u16gBackSpeedRailWayAxleToolValue := TO_UINT(((u16gBackSpeedRailWayAxle.Value - u16gBackSpeedRailWayAxle.AppScalingOffset) * u16gBackSpeedRailWayAxle.AppScalingDivisor / u16gBackSpeedRailWayAxle.AppScalingMultiplier * u16gBackSpeedRailWayAxle.ToolScalingMultiplier / u16gBackSpeedRailWayAxle.ToolScalingDivisor) + u16gBackSpeedRailWayAxle.ToolScalingOffset);

                  
END_GET
END_PROPERTY

PROPERTY u16gAvdvancePeriodToolValue : UINT
GET
                    IF u16gAvdvancePeriod.ToolScalingDivisor = 0 OR u16gAvdvancePeriod.AppScalingMultiplier = 0 THEN
	_MatchLog^.Error("Get u16gAvdvancePeriodToolValue", "Division by Zero!");
	RETURN;
END_IF

u16gAvdvancePeriodToolValue := TO_UINT(((u16gAvdvancePeriod.Value - u16gAvdvancePeriod.AppScalingOffset) * u16gAvdvancePeriod.AppScalingDivisor / u16gAvdvancePeriod.AppScalingMultiplier * u16gAvdvancePeriod.ToolScalingMultiplier / u16gAvdvancePeriod.ToolScalingDivisor) + u16gAvdvancePeriod.ToolScalingOffset);

                  
END_GET
END_PROPERTY

PROPERTY u16gPressureEfficiencyRateToolValue : UINT
GET
                    IF u16gPressureEfficiencyRate.ToolScalingDivisor = 0 OR u16gPressureEfficiencyRate.AppScalingMultiplier = 0 THEN
	_MatchLog^.Error("Get u16gPressureEfficiencyRateToolValue", "Division by Zero!");
	RETURN;
END_IF

u16gPressureEfficiencyRateToolValue := TO_UINT(((u16gPressureEfficiencyRate.Value - u16gPressureEfficiencyRate.AppScalingOffset) * u16gPressureEfficiencyRate.AppScalingDivisor / u16gPressureEfficiencyRate.AppScalingMultiplier * u16gPressureEfficiencyRate.ToolScalingMultiplier / u16gPressureEfficiencyRate.ToolScalingDivisor) + u16gPressureEfficiencyRate.ToolScalingOffset);

                  
END_GET
END_PROPERTY

METHOD InitializeCanSignals
                  u16gFrontSpeedRailWayAxle.AppScalingDivisor :=1;
u16gFrontSpeedRailWayAxle.AppScalingMultiplier :=1;
u16gFrontSpeedRailWayAxle.AppScalingOffset :=0;
u16gFrontSpeedRailWayAxle.AppUnit :="";
u16gFrontSpeedRailWayAxle.CanDefault :=0;
u16gFrontSpeedRailWayAxle.CanInit :=0;
u16gFrontSpeedRailWayAxle.CanMax :=VBasic.LibConst.U16_MAX;
u16gFrontSpeedRailWayAxle.CanMin :=VBasic.LibConst.U16_MIN;
u16gFrontSpeedRailWayAxle.CanUnit :="";
u16gFrontSpeedRailWayAxle.Description :="Front Speed Railway Axle in Km/h (A24)";
u16gFrontSpeedRailWayAxle.ErrorReaction := eErrorReaction.ERSIG_DFLT;
u16gFrontSpeedRailWayAxle.ReceiverAdress :=1;
u16gFrontSpeedRailWayAxle.ToolScalingDivisor :=1;
u16gFrontSpeedRailWayAxle.ToolScalingMultiplier :=1;
u16gFrontSpeedRailWayAxle.ToolScalingOffset :=0;
u16gFrontSpeedRailWayAxle.ToolUnit :="";

u16gBackSpeedRailWayAxle.AppScalingDivisor :=1;
u16gBackSpeedRailWayAxle.AppScalingMultiplier :=1;
u16gBackSpeedRailWayAxle.AppScalingOffset :=0;
u16gBackSpeedRailWayAxle.AppUnit :="";
u16gBackSpeedRailWayAxle.CanDefault :=0;
u16gBackSpeedRailWayAxle.CanInit :=0;
u16gBackSpeedRailWayAxle.CanMax :=VBasic.LibConst.U16_MAX;
u16gBackSpeedRailWayAxle.CanMin :=VBasic.LibConst.U16_MIN;
u16gBackSpeedRailWayAxle.CanUnit :="";
u16gBackSpeedRailWayAxle.Description :="Back Speed Railway Axle in Km/h";
u16gBackSpeedRailWayAxle.ErrorReaction := eErrorReaction.ERSIG_DFLT;
u16gBackSpeedRailWayAxle.ReceiverAdress :=1;
u16gBackSpeedRailWayAxle.ToolScalingDivisor :=1;
u16gBackSpeedRailWayAxle.ToolScalingMultiplier :=1;
u16gBackSpeedRailWayAxle.ToolScalingOffset :=0;
u16gBackSpeedRailWayAxle.ToolUnit :="";

u16gAvdvancePeriod.AppScalingDivisor :=1;
u16gAvdvancePeriod.AppScalingMultiplier :=1;
u16gAvdvancePeriod.AppScalingOffset :=0;
u16gAvdvancePeriod.AppUnit :="";
u16gAvdvancePeriod.CanDefault :=0;
u16gAvdvancePeriod.CanInit :=0;
u16gAvdvancePeriod.CanMax :=VBasic.LibConst.U16_MAX;
u16gAvdvancePeriod.CanMin :=VBasic.LibConst.U16_MIN;
u16gAvdvancePeriod.CanUnit :="";
u16gAvdvancePeriod.Description :="new signal";
u16gAvdvancePeriod.ErrorReaction := eErrorReaction.ERSIG_DFLT;
u16gAvdvancePeriod.ReceiverAdress :=1;
u16gAvdvancePeriod.ToolScalingDivisor :=1;
u16gAvdvancePeriod.ToolScalingMultiplier :=1;
u16gAvdvancePeriod.ToolScalingOffset :=0;
u16gAvdvancePeriod.ToolUnit :="";

u16gPressureEfficiencyRate.AppScalingDivisor :=1;
u16gPressureEfficiencyRate.AppScalingMultiplier :=1;
u16gPressureEfficiencyRate.AppScalingOffset :=0;
u16gPressureEfficiencyRate.AppUnit :="";
u16gPressureEfficiencyRate.CanDefault :=0;
u16gPressureEfficiencyRate.CanInit :=0;
u16gPressureEfficiencyRate.CanMax :=VBasic.LibConst.U16_MAX;
u16gPressureEfficiencyRate.CanMin :=VBasic.LibConst.U16_MIN;
u16gPressureEfficiencyRate.CanUnit :="";
u16gPressureEfficiencyRate.Description :="new signal";
u16gPressureEfficiencyRate.ErrorReaction := eErrorReaction.ERSIG_DFLT;
u16gPressureEfficiencyRate.ReceiverAdress :=1;
u16gPressureEfficiencyRate.ToolScalingDivisor :=1;
u16gPressureEfficiencyRate.ToolScalingMultiplier :=1;
u16gPressureEfficiencyRate.ToolScalingOffset :=0;
u16gPressureEfficiencyRate.ToolUnit :="";


                
END_METHOD
END_FUNCTION_BLOCK

FUNCTION_BLOCK Msg4C0SendToEvision7MessageClass EXTENDS CanReceiveMessageClass
  VAR_INPUT
    u16gForwardPumpCurrent : UInt16CanSignalClass;
    u16gBackwardPumpCurrent : UInt16CanSignalClass;
    i16gTrans1PressureSensorValue : Int16CanSignalClass;
    i16gTrans2PressureSensorValue : Int16CanSignalClass;
    Counter : UInt32CanSignalClass;
  END_VAR

            
          

METHOD SetData
  VAR_INPUT
    CanMsgPointer : POINTER TO CanMessageClass;
  END_VAR
                  IF IsValidPointer(canMsgPointer,'SetData') THEN
	SUPER^.SetData(CanMsgPointer);
	//Set the new data
	u16gForwardPumpCurrent.Value := canMsgPointer^.GetUint16(0);
	u16gBackwardPumpCurrent.Value := canMsgPointer^.GetUint16(16);
	i16gTrans1PressureSensorValue.Value := canMsgPointer^.GetInt16(32);
	i16gTrans2PressureSensorValue.Value := canMsgPointer^.GetInt16(48);
	//And increase the counter
	Counter.Value := CanMsgPointer^.Counter.Value;
END_IF

                
END_METHOD

PROPERTY u16gForwardPumpCurrentRawValue : UINT
GET
                    IF u16gForwardPumpCurrent.AppScalingMultiplier = 0 THEN
	_MatchLog^.Error("Get u16gForwardPumpCurrentRawValue", "Division by Zero!");
	RETURN;
End_IF

u16gForwardPumpCurrentRawValue := TO_UINT((u16gForwardPumpCurrent.Value - u16gForwardPumpCurrent.AppScalingOffset) * u16gForwardPumpCurrent.AppScalingDivisor / u16gForwardPumpCurrent.AppScalingMultiplier);

                  
END_GET
END_PROPERTY

PROPERTY u16gBackwardPumpCurrentRawValue : UINT
GET
                    IF u16gBackwardPumpCurrent.AppScalingMultiplier = 0 THEN
	_MatchLog^.Error("Get u16gBackwardPumpCurrentRawValue", "Division by Zero!");
	RETURN;
End_IF

u16gBackwardPumpCurrentRawValue := TO_UINT((u16gBackwardPumpCurrent.Value - u16gBackwardPumpCurrent.AppScalingOffset) * u16gBackwardPumpCurrent.AppScalingDivisor / u16gBackwardPumpCurrent.AppScalingMultiplier);

                  
END_GET
END_PROPERTY

PROPERTY i16gTrans1PressureSensorValueRawValue : INT
GET
                    IF i16gTrans1PressureSensorValue.AppScalingMultiplier = 0 THEN
	_MatchLog^.Error("Get i16gTrans1PressureSensorValueRawValue", "Division by Zero!");
	RETURN;
End_IF

i16gTrans1PressureSensorValueRawValue := TO_INT((i16gTrans1PressureSensorValue.Value - i16gTrans1PressureSensorValue.AppScalingOffset) * i16gTrans1PressureSensorValue.AppScalingDivisor / i16gTrans1PressureSensorValue.AppScalingMultiplier);

                  
END_GET
END_PROPERTY

PROPERTY i16gTrans2PressureSensorValueRawValue : INT
GET
                    IF i16gTrans2PressureSensorValue.AppScalingMultiplier = 0 THEN
	_MatchLog^.Error("Get i16gTrans2PressureSensorValueRawValue", "Division by Zero!");
	RETURN;
End_IF

i16gTrans2PressureSensorValueRawValue := TO_INT((i16gTrans2PressureSensorValue.Value - i16gTrans2PressureSensorValue.AppScalingOffset) * i16gTrans2PressureSensorValue.AppScalingDivisor / i16gTrans2PressureSensorValue.AppScalingMultiplier);

                  
END_GET
END_PROPERTY

PROPERTY u16gForwardPumpCurrentToolValue : UINT
GET
                    IF u16gForwardPumpCurrent.ToolScalingDivisor = 0 OR u16gForwardPumpCurrent.AppScalingMultiplier = 0 THEN
	_MatchLog^.Error("Get u16gForwardPumpCurrentToolValue", "Division by Zero!");
	RETURN;
END_IF

u16gForwardPumpCurrentToolValue := TO_UINT(((u16gForwardPumpCurrent.Value - u16gForwardPumpCurrent.AppScalingOffset) * u16gForwardPumpCurrent.AppScalingDivisor / u16gForwardPumpCurrent.AppScalingMultiplier * u16gForwardPumpCurrent.ToolScalingMultiplier / u16gForwardPumpCurrent.ToolScalingDivisor) + u16gForwardPumpCurrent.ToolScalingOffset);

                  
END_GET
END_PROPERTY

PROPERTY u16gBackwardPumpCurrentToolValue : UINT
GET
                    IF u16gBackwardPumpCurrent.ToolScalingDivisor = 0 OR u16gBackwardPumpCurrent.AppScalingMultiplier = 0 THEN
	_MatchLog^.Error("Get u16gBackwardPumpCurrentToolValue", "Division by Zero!");
	RETURN;
END_IF

u16gBackwardPumpCurrentToolValue := TO_UINT(((u16gBackwardPumpCurrent.Value - u16gBackwardPumpCurrent.AppScalingOffset) * u16gBackwardPumpCurrent.AppScalingDivisor / u16gBackwardPumpCurrent.AppScalingMultiplier * u16gBackwardPumpCurrent.ToolScalingMultiplier / u16gBackwardPumpCurrent.ToolScalingDivisor) + u16gBackwardPumpCurrent.ToolScalingOffset);

                  
END_GET
END_PROPERTY

PROPERTY i16gTrans1PressureSensorValueToolValue : INT
GET
                    IF i16gTrans1PressureSensorValue.ToolScalingDivisor = 0 OR i16gTrans1PressureSensorValue.AppScalingMultiplier = 0 THEN
	_MatchLog^.Error("Get i16gTrans1PressureSensorValueToolValue", "Division by Zero!");
	RETURN;
END_IF

i16gTrans1PressureSensorValueToolValue := TO_INT(((i16gTrans1PressureSensorValue.Value - i16gTrans1PressureSensorValue.AppScalingOffset) * i16gTrans1PressureSensorValue.AppScalingDivisor / i16gTrans1PressureSensorValue.AppScalingMultiplier * i16gTrans1PressureSensorValue.ToolScalingMultiplier / i16gTrans1PressureSensorValue.ToolScalingDivisor) + i16gTrans1PressureSensorValue.ToolScalingOffset);

                  
END_GET
END_PROPERTY

PROPERTY i16gTrans2PressureSensorValueToolValue : INT
GET
                    IF i16gTrans2PressureSensorValue.ToolScalingDivisor = 0 OR i16gTrans2PressureSensorValue.AppScalingMultiplier = 0 THEN
	_MatchLog^.Error("Get i16gTrans2PressureSensorValueToolValue", "Division by Zero!");
	RETURN;
END_IF

i16gTrans2PressureSensorValueToolValue := TO_INT(((i16gTrans2PressureSensorValue.Value - i16gTrans2PressureSensorValue.AppScalingOffset) * i16gTrans2PressureSensorValue.AppScalingDivisor / i16gTrans2PressureSensorValue.AppScalingMultiplier * i16gTrans2PressureSensorValue.ToolScalingMultiplier / i16gTrans2PressureSensorValue.ToolScalingDivisor) + i16gTrans2PressureSensorValue.ToolScalingOffset);

                  
END_GET
END_PROPERTY

METHOD InitializeCanSignals
                  u16gForwardPumpCurrent.AppScalingDivisor :=1;
u16gForwardPumpCurrent.AppScalingMultiplier :=1;
u16gForwardPumpCurrent.AppScalingOffset :=0;
u16gForwardPumpCurrent.AppUnit :="";
u16gForwardPumpCurrent.CanDefault :=0;
u16gForwardPumpCurrent.CanInit :=0;
u16gForwardPumpCurrent.CanMax :=VBasic.LibConst.U16_MAX;
u16gForwardPumpCurrent.CanMin :=VBasic.LibConst.U16_MIN;
u16gForwardPumpCurrent.CanUnit :="";
u16gForwardPumpCurrent.Description :="Pressure transmission 1";
u16gForwardPumpCurrent.ErrorReaction := eErrorReaction.ERSIG_DFLT;
u16gForwardPumpCurrent.ReceiverAdress :=1;
u16gForwardPumpCurrent.ToolScalingDivisor :=1;
u16gForwardPumpCurrent.ToolScalingMultiplier :=1;
u16gForwardPumpCurrent.ToolScalingOffset :=0;
u16gForwardPumpCurrent.ToolUnit :="";

u16gBackwardPumpCurrent.AppScalingDivisor :=1;
u16gBackwardPumpCurrent.AppScalingMultiplier :=1;
u16gBackwardPumpCurrent.AppScalingOffset :=0;
u16gBackwardPumpCurrent.AppUnit :="";
u16gBackwardPumpCurrent.CanDefault :=0;
u16gBackwardPumpCurrent.CanInit :=0;
u16gBackwardPumpCurrent.CanMax :=VBasic.LibConst.U16_MAX;
u16gBackwardPumpCurrent.CanMin :=VBasic.LibConst.U16_MIN;
u16gBackwardPumpCurrent.CanUnit :="";
u16gBackwardPumpCurrent.Description :="Pressure transmission 2";
u16gBackwardPumpCurrent.ErrorReaction := eErrorReaction.ERSIG_DFLT;
u16gBackwardPumpCurrent.ReceiverAdress :=1;
u16gBackwardPumpCurrent.ToolScalingDivisor :=1;
u16gBackwardPumpCurrent.ToolScalingMultiplier :=1;
u16gBackwardPumpCurrent.ToolScalingOffset :=0;
u16gBackwardPumpCurrent.ToolUnit :="";

i16gTrans1PressureSensorValue.AppScalingDivisor :=1;
i16gTrans1PressureSensorValue.AppScalingMultiplier :=1;
i16gTrans1PressureSensorValue.AppScalingOffset :=0;
i16gTrans1PressureSensorValue.AppUnit :="";
i16gTrans1PressureSensorValue.CanDefault :=0;
i16gTrans1PressureSensorValue.CanInit :=0;
i16gTrans1PressureSensorValue.CanMax :=VBasic.LibConst.I16_MAX;
i16gTrans1PressureSensorValue.CanMin :=VBasic.LibConst.I16_MIN;
i16gTrans1PressureSensorValue.CanUnit :="";
i16gTrans1PressureSensorValue.Description :="new signal";
i16gTrans1PressureSensorValue.ErrorReaction := eErrorReaction.ERSIG_DFLT;
i16gTrans1PressureSensorValue.ReceiverAdress :=1;
i16gTrans1PressureSensorValue.ToolScalingDivisor :=1;
i16gTrans1PressureSensorValue.ToolScalingMultiplier :=1;
i16gTrans1PressureSensorValue.ToolScalingOffset :=0;
i16gTrans1PressureSensorValue.ToolUnit :="";

i16gTrans2PressureSensorValue.AppScalingDivisor :=1;
i16gTrans2PressureSensorValue.AppScalingMultiplier :=1;
i16gTrans2PressureSensorValue.AppScalingOffset :=0;
i16gTrans2PressureSensorValue.AppUnit :="";
i16gTrans2PressureSensorValue.CanDefault :=0;
i16gTrans2PressureSensorValue.CanInit :=0;
i16gTrans2PressureSensorValue.CanMax :=VBasic.LibConst.I16_MAX;
i16gTrans2PressureSensorValue.CanMin :=VBasic.LibConst.I16_MIN;
i16gTrans2PressureSensorValue.CanUnit :="";
i16gTrans2PressureSensorValue.Description :="new signal";
i16gTrans2PressureSensorValue.ErrorReaction := eErrorReaction.ERSIG_DFLT;
i16gTrans2PressureSensorValue.ReceiverAdress :=1;
i16gTrans2PressureSensorValue.ToolScalingDivisor :=1;
i16gTrans2PressureSensorValue.ToolScalingMultiplier :=1;
i16gTrans2PressureSensorValue.ToolScalingOffset :=0;
i16gTrans2PressureSensorValue.ToolUnit :="";


                
END_METHOD
END_FUNCTION_BLOCK

FUNCTION_BLOCK Msg5C0SendToEvision7MessageClass EXTENDS CanReceiveMessageClass
  VAR_INPUT
    boAbutementNacelleTrackSide : BoolCanSignalClass;
    boAbutementNacelleCenteredSide : BoolCanSignalClass;
    boBasketTurretLimitation : BoolCanSignalClass;
    boPin217Fault : BoolCanSignalClass;
    boPin230Fault : BoolCanSignalClass;
    boPin243Fault : BoolCanSignalClass;
    boPin244Fault : BoolCanSignalClass;
    boPin245Fault : BoolCanSignalClass;
    boPin256Fault : BoolCanSignalClass;
    boPin257Fault : BoolCanSignalClass;
    boPin258Fault : BoolCanSignalClass;
    boPin103Fault : BoolCanSignalClass;
    boPin127Fault : BoolCanSignalClass;
    boPin104Fault : BoolCanSignalClass;
    boPin128Fault : BoolCanSignalClass;
    boPin105Fault : BoolCanSignalClass;
    boPin129Fault : BoolCanSignalClass;
    boPin106Fault : BoolCanSignalClass;
    boPin130Fault : BoolCanSignalClass;
    boPin107Fault : BoolCanSignalClass;
    boPin131Fault : BoolCanSignalClass;
    boPin108Fault : BoolCanSignalClass;
    boPin132Fault : BoolCanSignalClass;
    boPin109Fault : BoolCanSignalClass;
    boPin133Fault : BoolCanSignalClass;
    boPin110Fault : BoolCanSignalClass;
    boPin134Fault : BoolCanSignalClass;
    boPin111Fault : BoolCanSignalClass;
    boPin135Fault : BoolCanSignalClass;
    boPin112Fault : BoolCanSignalClass;
    boPin136Fault : BoolCanSignalClass;
    boPin113Fault : BoolCanSignalClass;
    boPin137Fault : BoolCanSignalClass;
    boPin114Fault : BoolCanSignalClass;
    boPin138Fault : BoolCanSignalClass;
    boPin115Fault : BoolCanSignalClass;
    boPin139Fault : BoolCanSignalClass;
    boPin116Fault : BoolCanSignalClass;
    boPin140Fault : BoolCanSignalClass;
    boPin117Fault : BoolCanSignalClass;
    boPin141Fault : BoolCanSignalClass;
    boPin122Fault : BoolCanSignalClass;
    boPin146Fault : BoolCanSignalClass;
    boPin123Fault : BoolCanSignalClass;
    boPin147Fault : BoolCanSignalClass;
    boPin124Fault : BoolCanSignalClass;
    boPin148Fault : BoolCanSignalClass;
    boPin153Fault : BoolCanSignalClass;
    boPin177Fault : BoolCanSignalClass;
    boPin156Fault : BoolCanSignalClass;
    boPin180Fault : BoolCanSignalClass;
    boPin159Fault : BoolCanSignalClass;
    boPin183Fault : BoolCanSignalClass;
    boPin186Fault : BoolCanSignalClass;
    boPin162Fault : BoolCanSignalClass;
    boPin189Fault : BoolCanSignalClass;
    boPin165Fault : BoolCanSignalClass;
    boPin192Fault : BoolCanSignalClass;
    boPin168Fault : BoolCanSignalClass;
    boPin195Fault : BoolCanSignalClass;
    boPin171Fault : BoolCanSignalClass;
    boPin154Fault : BoolCanSignalClass;
    boPin178Fault : BoolCanSignalClass;
    boPin157Fault : BoolCanSignalClass;
    Counter : UInt32CanSignalClass;
  END_VAR

            
          

METHOD SetData
  VAR_INPUT
    CanMsgPointer : POINTER TO CanMessageClass;
  END_VAR
                  IF IsValidPointer(canMsgPointer,'SetData') THEN
	SUPER^.SetData(CanMsgPointer);
	//Set the new data
	boAbutementNacelleTrackSide.Value := canMsgPointer^.GetBoolOnBit(0);
	boAbutementNacelleCenteredSide.Value := canMsgPointer^.GetBoolOnBit(1);
	boBasketTurretLimitation.Value := canMsgPointer^.GetBoolOnBit(2);
	boPin217Fault.Value := canMsgPointer^.GetBoolOnBit(3);
	boPin230Fault.Value := canMsgPointer^.GetBoolOnBit(4);
	boPin243Fault.Value := canMsgPointer^.GetBoolOnBit(5);
	boPin244Fault.Value := canMsgPointer^.GetBoolOnBit(6);
	boPin245Fault.Value := canMsgPointer^.GetBoolOnBit(7);
	boPin256Fault.Value := canMsgPointer^.GetBoolOnBit(8);
	boPin257Fault.Value := canMsgPointer^.GetBoolOnBit(9);
	boPin258Fault.Value := canMsgPointer^.GetBoolOnBit(10);
	boPin103Fault.Value := canMsgPointer^.GetBoolOnBit(11);
	boPin127Fault.Value := canMsgPointer^.GetBoolOnBit(12);
	boPin104Fault.Value := canMsgPointer^.GetBoolOnBit(13);
	boPin128Fault.Value := canMsgPointer^.GetBoolOnBit(14);
	boPin105Fault.Value := canMsgPointer^.GetBoolOnBit(15);
	boPin129Fault.Value := canMsgPointer^.GetBoolOnBit(16);
	boPin106Fault.Value := canMsgPointer^.GetBoolOnBit(17);
	boPin130Fault.Value := canMsgPointer^.GetBoolOnBit(18);
	boPin107Fault.Value := canMsgPointer^.GetBoolOnBit(19);
	boPin131Fault.Value := canMsgPointer^.GetBoolOnBit(20);
	boPin108Fault.Value := canMsgPointer^.GetBoolOnBit(21);
	boPin132Fault.Value := canMsgPointer^.GetBoolOnBit(22);
	boPin109Fault.Value := canMsgPointer^.GetBoolOnBit(23);
	boPin133Fault.Value := canMsgPointer^.GetBoolOnBit(24);
	boPin110Fault.Value := canMsgPointer^.GetBoolOnBit(25);
	boPin134Fault.Value := canMsgPointer^.GetBoolOnBit(26);
	boPin111Fault.Value := canMsgPointer^.GetBoolOnBit(27);
	boPin135Fault.Value := canMsgPointer^.GetBoolOnBit(28);
	boPin112Fault.Value := canMsgPointer^.GetBoolOnBit(29);
	boPin136Fault.Value := canMsgPointer^.GetBoolOnBit(30);
	boPin113Fault.Value := canMsgPointer^.GetBoolOnBit(31);
	boPin137Fault.Value := canMsgPointer^.GetBoolOnBit(32);
	boPin114Fault.Value := canMsgPointer^.GetBoolOnBit(33);
	boPin138Fault.Value := canMsgPointer^.GetBoolOnBit(34);
	boPin115Fault.Value := canMsgPointer^.GetBoolOnBit(35);
	boPin139Fault.Value := canMsgPointer^.GetBoolOnBit(36);
	boPin116Fault.Value := canMsgPointer^.GetBoolOnBit(37);
	boPin140Fault.Value := canMsgPointer^.GetBoolOnBit(38);
	boPin117Fault.Value := canMsgPointer^.GetBoolOnBit(39);
	boPin141Fault.Value := canMsgPointer^.GetBoolOnBit(40);
	boPin122Fault.Value := canMsgPointer^.GetBoolOnBit(41);
	boPin146Fault.Value := canMsgPointer^.GetBoolOnBit(42);
	boPin123Fault.Value := canMsgPointer^.GetBoolOnBit(43);
	boPin147Fault.Value := canMsgPointer^.GetBoolOnBit(44);
	boPin124Fault.Value := canMsgPointer^.GetBoolOnBit(45);
	boPin148Fault.Value := canMsgPointer^.GetBoolOnBit(46);
	boPin153Fault.Value := canMsgPointer^.GetBoolOnBit(47);
	boPin177Fault.Value := canMsgPointer^.GetBoolOnBit(48);
	boPin156Fault.Value := canMsgPointer^.GetBoolOnBit(49);
	boPin180Fault.Value := canMsgPointer^.GetBoolOnBit(50);
	boPin159Fault.Value := canMsgPointer^.GetBoolOnBit(51);
	boPin183Fault.Value := canMsgPointer^.GetBoolOnBit(52);
	boPin186Fault.Value := canMsgPointer^.GetBoolOnBit(53);
	boPin162Fault.Value := canMsgPointer^.GetBoolOnBit(54);
	boPin189Fault.Value := canMsgPointer^.GetBoolOnBit(55);
	boPin165Fault.Value := canMsgPointer^.GetBoolOnBit(56);
	boPin192Fault.Value := canMsgPointer^.GetBoolOnBit(57);
	boPin168Fault.Value := canMsgPointer^.GetBoolOnBit(58);
	boPin195Fault.Value := canMsgPointer^.GetBoolOnBit(59);
	boPin171Fault.Value := canMsgPointer^.GetBoolOnBit(60);
	boPin154Fault.Value := canMsgPointer^.GetBoolOnBit(61);
	boPin178Fault.Value := canMsgPointer^.GetBoolOnBit(62);
	boPin157Fault.Value := canMsgPointer^.GetBoolOnBit(63);
	//And increase the counter
	Counter.Value := CanMsgPointer^.Counter.Value;
END_IF

                
END_METHOD

PROPERTY boAbutementNacelleTrackSideRawValue : BOOL
GET
                    boAbutementNacelleTrackSideRawValue := boAbutementNacelleTrackSide.Value;

                  
END_GET
END_PROPERTY

PROPERTY boAbutementNacelleCenteredSideRawValue : BOOL
GET
                    boAbutementNacelleCenteredSideRawValue := boAbutementNacelleCenteredSide.Value;

                  
END_GET
END_PROPERTY

PROPERTY boBasketTurretLimitationRawValue : BOOL
GET
                    boBasketTurretLimitationRawValue := boBasketTurretLimitation.Value;

                  
END_GET
END_PROPERTY

PROPERTY boPin217FaultRawValue : BOOL
GET
                    boPin217FaultRawValue := boPin217Fault.Value;

                  
END_GET
END_PROPERTY

PROPERTY boPin230FaultRawValue : BOOL
GET
                    boPin230FaultRawValue := boPin230Fault.Value;

                  
END_GET
END_PROPERTY

PROPERTY boPin243FaultRawValue : BOOL
GET
                    boPin243FaultRawValue := boPin243Fault.Value;

                  
END_GET
END_PROPERTY

PROPERTY boPin244FaultRawValue : BOOL
GET
                    boPin244FaultRawValue := boPin244Fault.Value;

                  
END_GET
END_PROPERTY

PROPERTY boPin245FaultRawValue : BOOL
GET
                    boPin245FaultRawValue := boPin245Fault.Value;

                  
END_GET
END_PROPERTY

PROPERTY boPin256FaultRawValue : BOOL
GET
                    boPin256FaultRawValue := boPin256Fault.Value;

                  
END_GET
END_PROPERTY

PROPERTY boPin257FaultRawValue : BOOL
GET
                    boPin257FaultRawValue := boPin257Fault.Value;

                  
END_GET
END_PROPERTY

PROPERTY boPin258FaultRawValue : BOOL
GET
                    boPin258FaultRawValue := boPin258Fault.Value;

                  
END_GET
END_PROPERTY

PROPERTY boPin103FaultRawValue : BOOL
GET
                    boPin103FaultRawValue := boPin103Fault.Value;

                  
END_GET
END_PROPERTY

PROPERTY boPin127FaultRawValue : BOOL
GET
                    boPin127FaultRawValue := boPin127Fault.Value;

                  
END_GET
END_PROPERTY

PROPERTY boPin104FaultRawValue : BOOL
GET
                    boPin104FaultRawValue := boPin104Fault.Value;

                  
END_GET
END_PROPERTY

PROPERTY boPin128FaultRawValue : BOOL
GET
                    boPin128FaultRawValue := boPin128Fault.Value;

                  
END_GET
END_PROPERTY

PROPERTY boPin105FaultRawValue : BOOL
GET
                    boPin105FaultRawValue := boPin105Fault.Value;

                  
END_GET
END_PROPERTY

PROPERTY boPin129FaultRawValue : BOOL
GET
                    boPin129FaultRawValue := boPin129Fault.Value;

                  
END_GET
END_PROPERTY

PROPERTY boPin106FaultRawValue : BOOL
GET
                    boPin106FaultRawValue := boPin106Fault.Value;

                  
END_GET
END_PROPERTY

PROPERTY boPin130FaultRawValue : BOOL
GET
                    boPin130FaultRawValue := boPin130Fault.Value;

                  
END_GET
END_PROPERTY

PROPERTY boPin107FaultRawValue : BOOL
GET
                    boPin107FaultRawValue := boPin107Fault.Value;

                  
END_GET
END_PROPERTY

PROPERTY boPin131FaultRawValue : BOOL
GET
                    boPin131FaultRawValue := boPin131Fault.Value;

                  
END_GET
END_PROPERTY

PROPERTY boPin108FaultRawValue : BOOL
GET
                    boPin108FaultRawValue := boPin108Fault.Value;

                  
END_GET
END_PROPERTY

PROPERTY boPin132FaultRawValue : BOOL
GET
                    boPin132FaultRawValue := boPin132Fault.Value;

                  
END_GET
END_PROPERTY

PROPERTY boPin109FaultRawValue : BOOL
GET
                    boPin109FaultRawValue := boPin109Fault.Value;

                  
END_GET
END_PROPERTY

PROPERTY boPin133FaultRawValue : BOOL
GET
                    boPin133FaultRawValue := boPin133Fault.Value;

                  
END_GET
END_PROPERTY

PROPERTY boPin110FaultRawValue : BOOL
GET
                    boPin110FaultRawValue := boPin110Fault.Value;

                  
END_GET
END_PROPERTY

PROPERTY boPin134FaultRawValue : BOOL
GET
                    boPin134FaultRawValue := boPin134Fault.Value;

                  
END_GET
END_PROPERTY

PROPERTY boPin111FaultRawValue : BOOL
GET
                    boPin111FaultRawValue := boPin111Fault.Value;

                  
END_GET
END_PROPERTY

PROPERTY boPin135FaultRawValue : BOOL
GET
                    boPin135FaultRawValue := boPin135Fault.Value;

                  
END_GET
END_PROPERTY

PROPERTY boPin112FaultRawValue : BOOL
GET
                    boPin112FaultRawValue := boPin112Fault.Value;

                  
END_GET
END_PROPERTY

PROPERTY boPin136FaultRawValue : BOOL
GET
                    boPin136FaultRawValue := boPin136Fault.Value;

                  
END_GET
END_PROPERTY

PROPERTY boPin113FaultRawValue : BOOL
GET
                    boPin113FaultRawValue := boPin113Fault.Value;

                  
END_GET
END_PROPERTY

PROPERTY boPin137FaultRawValue : BOOL
GET
                    boPin137FaultRawValue := boPin137Fault.Value;

                  
END_GET
END_PROPERTY

PROPERTY boPin114FaultRawValue : BOOL
GET
                    boPin114FaultRawValue := boPin114Fault.Value;

                  
END_GET
END_PROPERTY

PROPERTY boPin138FaultRawValue : BOOL
GET
                    boPin138FaultRawValue := boPin138Fault.Value;

                  
END_GET
END_PROPERTY

PROPERTY boPin115FaultRawValue : BOOL
GET
                    boPin115FaultRawValue := boPin115Fault.Value;

                  
END_GET
END_PROPERTY

PROPERTY boPin139FaultRawValue : BOOL
GET
                    boPin139FaultRawValue := boPin139Fault.Value;

                  
END_GET
END_PROPERTY

PROPERTY boPin116FaultRawValue : BOOL
GET
                    boPin116FaultRawValue := boPin116Fault.Value;

                  
END_GET
END_PROPERTY

PROPERTY boPin140FaultRawValue : BOOL
GET
                    boPin140FaultRawValue := boPin140Fault.Value;

                  
END_GET
END_PROPERTY

PROPERTY boPin117FaultRawValue : BOOL
GET
                    boPin117FaultRawValue := boPin117Fault.Value;

                  
END_GET
END_PROPERTY

PROPERTY boPin141FaultRawValue : BOOL
GET
                    boPin141FaultRawValue := boPin141Fault.Value;

                  
END_GET
END_PROPERTY

PROPERTY boPin122FaultRawValue : BOOL
GET
                    boPin122FaultRawValue := boPin122Fault.Value;

                  
END_GET
END_PROPERTY

PROPERTY boPin146FaultRawValue : BOOL
GET
                    boPin146FaultRawValue := boPin146Fault.Value;

                  
END_GET
END_PROPERTY

PROPERTY boPin123FaultRawValue : BOOL
GET
                    boPin123FaultRawValue := boPin123Fault.Value;

                  
END_GET
END_PROPERTY

PROPERTY boPin147FaultRawValue : BOOL
GET
                    boPin147FaultRawValue := boPin147Fault.Value;

                  
END_GET
END_PROPERTY

PROPERTY boPin124FaultRawValue : BOOL
GET
                    boPin124FaultRawValue := boPin124Fault.Value;

                  
END_GET
END_PROPERTY

PROPERTY boPin148FaultRawValue : BOOL
GET
                    boPin148FaultRawValue := boPin148Fault.Value;

                  
END_GET
END_PROPERTY

PROPERTY boPin153FaultRawValue : BOOL
GET
                    boPin153FaultRawValue := boPin153Fault.Value;

                  
END_GET
END_PROPERTY

PROPERTY boPin177FaultRawValue : BOOL
GET
                    boPin177FaultRawValue := boPin177Fault.Value;

                  
END_GET
END_PROPERTY

PROPERTY boPin156FaultRawValue : BOOL
GET
                    boPin156FaultRawValue := boPin156Fault.Value;

                  
END_GET
END_PROPERTY

PROPERTY boPin180FaultRawValue : BOOL
GET
                    boPin180FaultRawValue := boPin180Fault.Value;

                  
END_GET
END_PROPERTY

PROPERTY boPin159FaultRawValue : BOOL
GET
                    boPin159FaultRawValue := boPin159Fault.Value;

                  
END_GET
END_PROPERTY

PROPERTY boPin183FaultRawValue : BOOL
GET
                    boPin183FaultRawValue := boPin183Fault.Value;

                  
END_GET
END_PROPERTY

PROPERTY boPin186FaultRawValue : BOOL
GET
                    boPin186FaultRawValue := boPin186Fault.Value;

                  
END_GET
END_PROPERTY

PROPERTY boPin162FaultRawValue : BOOL
GET
                    boPin162FaultRawValue := boPin162Fault.Value;

                  
END_GET
END_PROPERTY

PROPERTY boPin189FaultRawValue : BOOL
GET
                    boPin189FaultRawValue := boPin189Fault.Value;

                  
END_GET
END_PROPERTY

PROPERTY boPin165FaultRawValue : BOOL
GET
                    boPin165FaultRawValue := boPin165Fault.Value;

                  
END_GET
END_PROPERTY

PROPERTY boPin192FaultRawValue : BOOL
GET
                    boPin192FaultRawValue := boPin192Fault.Value;

                  
END_GET
END_PROPERTY

PROPERTY boPin168FaultRawValue : BOOL
GET
                    boPin168FaultRawValue := boPin168Fault.Value;

                  
END_GET
END_PROPERTY

PROPERTY boPin195FaultRawValue : BOOL
GET
                    boPin195FaultRawValue := boPin195Fault.Value;

                  
END_GET
END_PROPERTY

PROPERTY boPin171FaultRawValue : BOOL
GET
                    boPin171FaultRawValue := boPin171Fault.Value;

                  
END_GET
END_PROPERTY

PROPERTY boPin154FaultRawValue : BOOL
GET
                    boPin154FaultRawValue := boPin154Fault.Value;

                  
END_GET
END_PROPERTY

PROPERTY boPin178FaultRawValue : BOOL
GET
                    boPin178FaultRawValue := boPin178Fault.Value;

                  
END_GET
END_PROPERTY

PROPERTY boPin157FaultRawValue : BOOL
GET
                    boPin157FaultRawValue := boPin157Fault.Value;

                  
END_GET
END_PROPERTY

PROPERTY boAbutementNacelleTrackSideToolValue : BOOL
GET
                    boAbutementNacelleTrackSideToolValue := boAbutementNacelleTrackSide.Value;

                  
END_GET
END_PROPERTY

PROPERTY boAbutementNacelleCenteredSideToolValue : BOOL
GET
                    boAbutementNacelleCenteredSideToolValue := boAbutementNacelleCenteredSide.Value;

                  
END_GET
END_PROPERTY

PROPERTY boBasketTurretLimitationToolValue : BOOL
GET
                    boBasketTurretLimitationToolValue := boBasketTurretLimitation.Value;

                  
END_GET
END_PROPERTY

PROPERTY boPin217FaultToolValue : BOOL
GET
                    boPin217FaultToolValue := boPin217Fault.Value;

                  
END_GET
END_PROPERTY

PROPERTY boPin230FaultToolValue : BOOL
GET
                    boPin230FaultToolValue := boPin230Fault.Value;

                  
END_GET
END_PROPERTY

PROPERTY boPin243FaultToolValue : BOOL
GET
                    boPin243FaultToolValue := boPin243Fault.Value;

                  
END_GET
END_PROPERTY

PROPERTY boPin244FaultToolValue : BOOL
GET
                    boPin244FaultToolValue := boPin244Fault.Value;

                  
END_GET
END_PROPERTY

PROPERTY boPin245FaultToolValue : BOOL
GET
                    boPin245FaultToolValue := boPin245Fault.Value;

                  
END_GET
END_PROPERTY

PROPERTY boPin256FaultToolValue : BOOL
GET
                    boPin256FaultToolValue := boPin256Fault.Value;

                  
END_GET
END_PROPERTY

PROPERTY boPin257FaultToolValue : BOOL
GET
                    boPin257FaultToolValue := boPin257Fault.Value;

                  
END_GET
END_PROPERTY

PROPERTY boPin258FaultToolValue : BOOL
GET
                    boPin258FaultToolValue := boPin258Fault.Value;

                  
END_GET
END_PROPERTY

PROPERTY boPin103FaultToolValue : BOOL
GET
                    boPin103FaultToolValue := boPin103Fault.Value;

                  
END_GET
END_PROPERTY

PROPERTY boPin127FaultToolValue : BOOL
GET
                    boPin127FaultToolValue := boPin127Fault.Value;

                  
END_GET
END_PROPERTY

PROPERTY boPin104FaultToolValue : BOOL
GET
                    boPin104FaultToolValue := boPin104Fault.Value;

                  
END_GET
END_PROPERTY

PROPERTY boPin128FaultToolValue : BOOL
GET
                    boPin128FaultToolValue := boPin128Fault.Value;

                  
END_GET
END_PROPERTY

PROPERTY boPin105FaultToolValue : BOOL
GET
                    boPin105FaultToolValue := boPin105Fault.Value;

                  
END_GET
END_PROPERTY

PROPERTY boPin129FaultToolValue : BOOL
GET
                    boPin129FaultToolValue := boPin129Fault.Value;

                  
END_GET
END_PROPERTY

PROPERTY boPin106FaultToolValue : BOOL
GET
                    boPin106FaultToolValue := boPin106Fault.Value;

                  
END_GET
END_PROPERTY

PROPERTY boPin130FaultToolValue : BOOL
GET
                    boPin130FaultToolValue := boPin130Fault.Value;

                  
END_GET
END_PROPERTY

PROPERTY boPin107FaultToolValue : BOOL
GET
                    boPin107FaultToolValue := boPin107Fault.Value;

                  
END_GET
END_PROPERTY

PROPERTY boPin131FaultToolValue : BOOL
GET
                    boPin131FaultToolValue := boPin131Fault.Value;

                  
END_GET
END_PROPERTY

PROPERTY boPin108FaultToolValue : BOOL
GET
                    boPin108FaultToolValue := boPin108Fault.Value;

                  
END_GET
END_PROPERTY

PROPERTY boPin132FaultToolValue : BOOL
GET
                    boPin132FaultToolValue := boPin132Fault.Value;

                  
END_GET
END_PROPERTY

PROPERTY boPin109FaultToolValue : BOOL
GET
                    boPin109FaultToolValue := boPin109Fault.Value;

                  
END_GET
END_PROPERTY

PROPERTY boPin133FaultToolValue : BOOL
GET
                    boPin133FaultToolValue := boPin133Fault.Value;

                  
END_GET
END_PROPERTY

PROPERTY boPin110FaultToolValue : BOOL
GET
                    boPin110FaultToolValue := boPin110Fault.Value;

                  
END_GET
END_PROPERTY

PROPERTY boPin134FaultToolValue : BOOL
GET
                    boPin134FaultToolValue := boPin134Fault.Value;

                  
END_GET
END_PROPERTY

PROPERTY boPin111FaultToolValue : BOOL
GET
                    boPin111FaultToolValue := boPin111Fault.Value;

                  
END_GET
END_PROPERTY

PROPERTY boPin135FaultToolValue : BOOL
GET
                    boPin135FaultToolValue := boPin135Fault.Value;

                  
END_GET
END_PROPERTY

PROPERTY boPin112FaultToolValue : BOOL
GET
                    boPin112FaultToolValue := boPin112Fault.Value;

                  
END_GET
END_PROPERTY

PROPERTY boPin136FaultToolValue : BOOL
GET
                    boPin136FaultToolValue := boPin136Fault.Value;

                  
END_GET
END_PROPERTY

PROPERTY boPin113FaultToolValue : BOOL
GET
                    boPin113FaultToolValue := boPin113Fault.Value;

                  
END_GET
END_PROPERTY

PROPERTY boPin137FaultToolValue : BOOL
GET
                    boPin137FaultToolValue := boPin137Fault.Value;

                  
END_GET
END_PROPERTY

PROPERTY boPin114FaultToolValue : BOOL
GET
                    boPin114FaultToolValue := boPin114Fault.Value;

                  
END_GET
END_PROPERTY

PROPERTY boPin138FaultToolValue : BOOL
GET
                    boPin138FaultToolValue := boPin138Fault.Value;

                  
END_GET
END_PROPERTY

PROPERTY boPin115FaultToolValue : BOOL
GET
                    boPin115FaultToolValue := boPin115Fault.Value;

                  
END_GET
END_PROPERTY

PROPERTY boPin139FaultToolValue : BOOL
GET
                    boPin139FaultToolValue := boPin139Fault.Value;

                  
END_GET
END_PROPERTY

PROPERTY boPin116FaultToolValue : BOOL
GET
                    boPin116FaultToolValue := boPin116Fault.Value;

                  
END_GET
END_PROPERTY

PROPERTY boPin140FaultToolValue : BOOL
GET
                    boPin140FaultToolValue := boPin140Fault.Value;

                  
END_GET
END_PROPERTY

PROPERTY boPin117FaultToolValue : BOOL
GET
                    boPin117FaultToolValue := boPin117Fault.Value;

                  
END_GET
END_PROPERTY

PROPERTY boPin141FaultToolValue : BOOL
GET
                    boPin141FaultToolValue := boPin141Fault.Value;

                  
END_GET
END_PROPERTY

PROPERTY boPin122FaultToolValue : BOOL
GET
                    boPin122FaultToolValue := boPin122Fault.Value;

                  
END_GET
END_PROPERTY

PROPERTY boPin146FaultToolValue : BOOL
GET
                    boPin146FaultToolValue := boPin146Fault.Value;

                  
END_GET
END_PROPERTY

PROPERTY boPin123FaultToolValue : BOOL
GET
                    boPin123FaultToolValue := boPin123Fault.Value;

                  
END_GET
END_PROPERTY

PROPERTY boPin147FaultToolValue : BOOL
GET
                    boPin147FaultToolValue := boPin147Fault.Value;

                  
END_GET
END_PROPERTY

PROPERTY boPin124FaultToolValue : BOOL
GET
                    boPin124FaultToolValue := boPin124Fault.Value;

                  
END_GET
END_PROPERTY

PROPERTY boPin148FaultToolValue : BOOL
GET
                    boPin148FaultToolValue := boPin148Fault.Value;

                  
END_GET
END_PROPERTY

PROPERTY boPin153FaultToolValue : BOOL
GET
                    boPin153FaultToolValue := boPin153Fault.Value;

                  
END_GET
END_PROPERTY

PROPERTY boPin177FaultToolValue : BOOL
GET
                    boPin177FaultToolValue := boPin177Fault.Value;

                  
END_GET
END_PROPERTY

PROPERTY boPin156FaultToolValue : BOOL
GET
                    boPin156FaultToolValue := boPin156Fault.Value;

                  
END_GET
END_PROPERTY

PROPERTY boPin180FaultToolValue : BOOL
GET
                    boPin180FaultToolValue := boPin180Fault.Value;

                  
END_GET
END_PROPERTY

PROPERTY boPin159FaultToolValue : BOOL
GET
                    boPin159FaultToolValue := boPin159Fault.Value;

                  
END_GET
END_PROPERTY

PROPERTY boPin183FaultToolValue : BOOL
GET
                    boPin183FaultToolValue := boPin183Fault.Value;

                  
END_GET
END_PROPERTY

PROPERTY boPin186FaultToolValue : BOOL
GET
                    boPin186FaultToolValue := boPin186Fault.Value;

                  
END_GET
END_PROPERTY

PROPERTY boPin162FaultToolValue : BOOL
GET
                    boPin162FaultToolValue := boPin162Fault.Value;

                  
END_GET
END_PROPERTY

PROPERTY boPin189FaultToolValue : BOOL
GET
                    boPin189FaultToolValue := boPin189Fault.Value;

                  
END_GET
END_PROPERTY

PROPERTY boPin165FaultToolValue : BOOL
GET
                    boPin165FaultToolValue := boPin165Fault.Value;

                  
END_GET
END_PROPERTY

PROPERTY boPin192FaultToolValue : BOOL
GET
                    boPin192FaultToolValue := boPin192Fault.Value;

                  
END_GET
END_PROPERTY

PROPERTY boPin168FaultToolValue : BOOL
GET
                    boPin168FaultToolValue := boPin168Fault.Value;

                  
END_GET
END_PROPERTY

PROPERTY boPin195FaultToolValue : BOOL
GET
                    boPin195FaultToolValue := boPin195Fault.Value;

                  
END_GET
END_PROPERTY

PROPERTY boPin171FaultToolValue : BOOL
GET
                    boPin171FaultToolValue := boPin171Fault.Value;

                  
END_GET
END_PROPERTY

PROPERTY boPin154FaultToolValue : BOOL
GET
                    boPin154FaultToolValue := boPin154Fault.Value;

                  
END_GET
END_PROPERTY

PROPERTY boPin178FaultToolValue : BOOL
GET
                    boPin178FaultToolValue := boPin178Fault.Value;

                  
END_GET
END_PROPERTY

PROPERTY boPin157FaultToolValue : BOOL
GET
                    boPin157FaultToolValue := boPin157Fault.Value;

                  
END_GET
END_PROPERTY

METHOD InitializeCanSignals
                  boAbutementNacelleTrackSide.AppScalingDivisor :=1;
boAbutementNacelleTrackSide.AppScalingMultiplier :=1;
boAbutementNacelleTrackSide.AppScalingOffset :=0;
boAbutementNacelleTrackSide.AppUnit :="";
boAbutementNacelleTrackSide.CanDefault :=0;
boAbutementNacelleTrackSide.CanInit :=0;
boAbutementNacelleTrackSide.CanMax :=1;
boAbutementNacelleTrackSide.CanMin :=0;
boAbutementNacelleTrackSide.CanUnit :="";
boAbutementNacelleTrackSide.Description :="for the Neotec diag pages";
boAbutementNacelleTrackSide.ErrorReaction := eErrorReaction.ERSIG_DFLT;
boAbutementNacelleTrackSide.ReceiverAdress :=1;
boAbutementNacelleTrackSide.ToolScalingDivisor :=1;
boAbutementNacelleTrackSide.ToolScalingMultiplier :=1;
boAbutementNacelleTrackSide.ToolScalingOffset :=0;
boAbutementNacelleTrackSide.ToolUnit :="";

boAbutementNacelleCenteredSide.AppScalingDivisor :=1;
boAbutementNacelleCenteredSide.AppScalingMultiplier :=1;
boAbutementNacelleCenteredSide.AppScalingOffset :=0;
boAbutementNacelleCenteredSide.AppUnit :="";
boAbutementNacelleCenteredSide.CanDefault :=0;
boAbutementNacelleCenteredSide.CanInit :=0;
boAbutementNacelleCenteredSide.CanMax :=1;
boAbutementNacelleCenteredSide.CanMin :=0;
boAbutementNacelleCenteredSide.CanUnit :="";
boAbutementNacelleCenteredSide.Description :="for the Neotec diag pages";
boAbutementNacelleCenteredSide.ErrorReaction := eErrorReaction.ERSIG_DFLT;
boAbutementNacelleCenteredSide.ReceiverAdress :=1;
boAbutementNacelleCenteredSide.ToolScalingDivisor :=1;
boAbutementNacelleCenteredSide.ToolScalingMultiplier :=1;
boAbutementNacelleCenteredSide.ToolScalingOffset :=0;
boAbutementNacelleCenteredSide.ToolUnit :="";

boBasketTurretLimitation.AppScalingDivisor :=1;
boBasketTurretLimitation.AppScalingMultiplier :=1;
boBasketTurretLimitation.AppScalingOffset :=0;
boBasketTurretLimitation.AppUnit :="";
boBasketTurretLimitation.CanDefault :=0;
boBasketTurretLimitation.CanInit :=0;
boBasketTurretLimitation.CanMax :=1;
boBasketTurretLimitation.CanMin :=0;
boBasketTurretLimitation.CanUnit :="";
boBasketTurretLimitation.Description :="for the Neotec diag pages";
boBasketTurretLimitation.ErrorReaction := eErrorReaction.ERSIG_DFLT;
boBasketTurretLimitation.ReceiverAdress :=1;
boBasketTurretLimitation.ToolScalingDivisor :=1;
boBasketTurretLimitation.ToolScalingMultiplier :=1;
boBasketTurretLimitation.ToolScalingOffset :=0;
boBasketTurretLimitation.ToolUnit :="";

boPin217Fault.AppScalingDivisor :=1;
boPin217Fault.AppScalingMultiplier :=1;
boPin217Fault.AppScalingOffset :=0;
boPin217Fault.AppUnit :="";
boPin217Fault.CanDefault :=0;
boPin217Fault.CanInit :=0;
boPin217Fault.CanMax :=1;
boPin217Fault.CanMin :=0;
boPin217Fault.CanUnit :="";
boPin217Fault.Description :="for the Neotec diag pages";
boPin217Fault.ErrorReaction := eErrorReaction.ERSIG_DFLT;
boPin217Fault.ReceiverAdress :=1;
boPin217Fault.ToolScalingDivisor :=1;
boPin217Fault.ToolScalingMultiplier :=1;
boPin217Fault.ToolScalingOffset :=0;
boPin217Fault.ToolUnit :="";

boPin230Fault.AppScalingDivisor :=1;
boPin230Fault.AppScalingMultiplier :=1;
boPin230Fault.AppScalingOffset :=0;
boPin230Fault.AppUnit :="";
boPin230Fault.CanDefault :=0;
boPin230Fault.CanInit :=0;
boPin230Fault.CanMax :=1;
boPin230Fault.CanMin :=0;
boPin230Fault.CanUnit :="";
boPin230Fault.Description :="for the Neotec diag pages";
boPin230Fault.ErrorReaction := eErrorReaction.ERSIG_DFLT;
boPin230Fault.ReceiverAdress :=1;
boPin230Fault.ToolScalingDivisor :=1;
boPin230Fault.ToolScalingMultiplier :=1;
boPin230Fault.ToolScalingOffset :=0;
boPin230Fault.ToolUnit :="";

boPin243Fault.AppScalingDivisor :=1;
boPin243Fault.AppScalingMultiplier :=1;
boPin243Fault.AppScalingOffset :=0;
boPin243Fault.AppUnit :="";
boPin243Fault.CanDefault :=0;
boPin243Fault.CanInit :=0;
boPin243Fault.CanMax :=1;
boPin243Fault.CanMin :=0;
boPin243Fault.CanUnit :="";
boPin243Fault.Description :="for the Neotec diag pages";
boPin243Fault.ErrorReaction := eErrorReaction.ERSIG_DFLT;
boPin243Fault.ReceiverAdress :=1;
boPin243Fault.ToolScalingDivisor :=1;
boPin243Fault.ToolScalingMultiplier :=1;
boPin243Fault.ToolScalingOffset :=0;
boPin243Fault.ToolUnit :="";

boPin244Fault.AppScalingDivisor :=1;
boPin244Fault.AppScalingMultiplier :=1;
boPin244Fault.AppScalingOffset :=0;
boPin244Fault.AppUnit :="";
boPin244Fault.CanDefault :=0;
boPin244Fault.CanInit :=0;
boPin244Fault.CanMax :=1;
boPin244Fault.CanMin :=0;
boPin244Fault.CanUnit :="";
boPin244Fault.Description :="for the Neotec diag pages";
boPin244Fault.ErrorReaction := eErrorReaction.ERSIG_DFLT;
boPin244Fault.ReceiverAdress :=1;
boPin244Fault.ToolScalingDivisor :=1;
boPin244Fault.ToolScalingMultiplier :=1;
boPin244Fault.ToolScalingOffset :=0;
boPin244Fault.ToolUnit :="";

boPin245Fault.AppScalingDivisor :=1;
boPin245Fault.AppScalingMultiplier :=1;
boPin245Fault.AppScalingOffset :=0;
boPin245Fault.AppUnit :="";
boPin245Fault.CanDefault :=0;
boPin245Fault.CanInit :=0;
boPin245Fault.CanMax :=1;
boPin245Fault.CanMin :=0;
boPin245Fault.CanUnit :="";
boPin245Fault.Description :="for the Neotec diag pages";
boPin245Fault.ErrorReaction := eErrorReaction.ERSIG_DFLT;
boPin245Fault.ReceiverAdress :=1;
boPin245Fault.ToolScalingDivisor :=1;
boPin245Fault.ToolScalingMultiplier :=1;
boPin245Fault.ToolScalingOffset :=0;
boPin245Fault.ToolUnit :="";

boPin256Fault.AppScalingDivisor :=1;
boPin256Fault.AppScalingMultiplier :=1;
boPin256Fault.AppScalingOffset :=0;
boPin256Fault.AppUnit :="";
boPin256Fault.CanDefault :=0;
boPin256Fault.CanInit :=0;
boPin256Fault.CanMax :=1;
boPin256Fault.CanMin :=0;
boPin256Fault.CanUnit :="";
boPin256Fault.Description :="for the Neotec diag pages";
boPin256Fault.ErrorReaction := eErrorReaction.ERSIG_DFLT;
boPin256Fault.ReceiverAdress :=1;
boPin256Fault.ToolScalingDivisor :=1;
boPin256Fault.ToolScalingMultiplier :=1;
boPin256Fault.ToolScalingOffset :=0;
boPin256Fault.ToolUnit :="";

boPin257Fault.AppScalingDivisor :=1;
boPin257Fault.AppScalingMultiplier :=1;
boPin257Fault.AppScalingOffset :=0;
boPin257Fault.AppUnit :="";
boPin257Fault.CanDefault :=0;
boPin257Fault.CanInit :=0;
boPin257Fault.CanMax :=1;
boPin257Fault.CanMin :=0;
boPin257Fault.CanUnit :="";
boPin257Fault.Description :="for the Neotec diag pages";
boPin257Fault.ErrorReaction := eErrorReaction.ERSIG_DFLT;
boPin257Fault.ReceiverAdress :=1;
boPin257Fault.ToolScalingDivisor :=1;
boPin257Fault.ToolScalingMultiplier :=1;
boPin257Fault.ToolScalingOffset :=0;
boPin257Fault.ToolUnit :="";

boPin258Fault.AppScalingDivisor :=1;
boPin258Fault.AppScalingMultiplier :=1;
boPin258Fault.AppScalingOffset :=0;
boPin258Fault.AppUnit :="";
boPin258Fault.CanDefault :=0;
boPin258Fault.CanInit :=0;
boPin258Fault.CanMax :=1;
boPin258Fault.CanMin :=0;
boPin258Fault.CanUnit :="";
boPin258Fault.Description :="for the Neotec diag pages";
boPin258Fault.ErrorReaction := eErrorReaction.ERSIG_DFLT;
boPin258Fault.ReceiverAdress :=1;
boPin258Fault.ToolScalingDivisor :=1;
boPin258Fault.ToolScalingMultiplier :=1;
boPin258Fault.ToolScalingOffset :=0;
boPin258Fault.ToolUnit :="";

boPin103Fault.AppScalingDivisor :=1;
boPin103Fault.AppScalingMultiplier :=1;
boPin103Fault.AppScalingOffset :=0;
boPin103Fault.AppUnit :="";
boPin103Fault.CanDefault :=0;
boPin103Fault.CanInit :=0;
boPin103Fault.CanMax :=1;
boPin103Fault.CanMin :=0;
boPin103Fault.CanUnit :="";
boPin103Fault.Description :="for the Neotec diag pages";
boPin103Fault.ErrorReaction := eErrorReaction.ERSIG_DFLT;
boPin103Fault.ReceiverAdress :=1;
boPin103Fault.ToolScalingDivisor :=1;
boPin103Fault.ToolScalingMultiplier :=1;
boPin103Fault.ToolScalingOffset :=0;
boPin103Fault.ToolUnit :="";

boPin127Fault.AppScalingDivisor :=1;
boPin127Fault.AppScalingMultiplier :=1;
boPin127Fault.AppScalingOffset :=0;
boPin127Fault.AppUnit :="";
boPin127Fault.CanDefault :=0;
boPin127Fault.CanInit :=0;
boPin127Fault.CanMax :=1;
boPin127Fault.CanMin :=0;
boPin127Fault.CanUnit :="";
boPin127Fault.Description :="for the Neotec diag pages";
boPin127Fault.ErrorReaction := eErrorReaction.ERSIG_DFLT;
boPin127Fault.ReceiverAdress :=1;
boPin127Fault.ToolScalingDivisor :=1;
boPin127Fault.ToolScalingMultiplier :=1;
boPin127Fault.ToolScalingOffset :=0;
boPin127Fault.ToolUnit :="";

boPin104Fault.AppScalingDivisor :=1;
boPin104Fault.AppScalingMultiplier :=1;
boPin104Fault.AppScalingOffset :=0;
boPin104Fault.AppUnit :="";
boPin104Fault.CanDefault :=0;
boPin104Fault.CanInit :=0;
boPin104Fault.CanMax :=1;
boPin104Fault.CanMin :=0;
boPin104Fault.CanUnit :="";
boPin104Fault.Description :="for the Neotec diag pages";
boPin104Fault.ErrorReaction := eErrorReaction.ERSIG_DFLT;
boPin104Fault.ReceiverAdress :=1;
boPin104Fault.ToolScalingDivisor :=1;
boPin104Fault.ToolScalingMultiplier :=1;
boPin104Fault.ToolScalingOffset :=0;
boPin104Fault.ToolUnit :="";

boPin128Fault.AppScalingDivisor :=1;
boPin128Fault.AppScalingMultiplier :=1;
boPin128Fault.AppScalingOffset :=0;
boPin128Fault.AppUnit :="";
boPin128Fault.CanDefault :=0;
boPin128Fault.CanInit :=0;
boPin128Fault.CanMax :=1;
boPin128Fault.CanMin :=0;
boPin128Fault.CanUnit :="";
boPin128Fault.Description :="for the Neotec diag pages";
boPin128Fault.ErrorReaction := eErrorReaction.ERSIG_DFLT;
boPin128Fault.ReceiverAdress :=1;
boPin128Fault.ToolScalingDivisor :=1;
boPin128Fault.ToolScalingMultiplier :=1;
boPin128Fault.ToolScalingOffset :=0;
boPin128Fault.ToolUnit :="";

boPin105Fault.AppScalingDivisor :=1;
boPin105Fault.AppScalingMultiplier :=1;
boPin105Fault.AppScalingOffset :=0;
boPin105Fault.AppUnit :="";
boPin105Fault.CanDefault :=0;
boPin105Fault.CanInit :=0;
boPin105Fault.CanMax :=1;
boPin105Fault.CanMin :=0;
boPin105Fault.CanUnit :="";
boPin105Fault.Description :="for the Neotec diag pages";
boPin105Fault.ErrorReaction := eErrorReaction.ERSIG_DFLT;
boPin105Fault.ReceiverAdress :=1;
boPin105Fault.ToolScalingDivisor :=1;
boPin105Fault.ToolScalingMultiplier :=1;
boPin105Fault.ToolScalingOffset :=0;
boPin105Fault.ToolUnit :="";

boPin129Fault.AppScalingDivisor :=1;
boPin129Fault.AppScalingMultiplier :=1;
boPin129Fault.AppScalingOffset :=0;
boPin129Fault.AppUnit :="";
boPin129Fault.CanDefault :=0;
boPin129Fault.CanInit :=0;
boPin129Fault.CanMax :=1;
boPin129Fault.CanMin :=0;
boPin129Fault.CanUnit :="";
boPin129Fault.Description :="for the Neotec diag pages";
boPin129Fault.ErrorReaction := eErrorReaction.ERSIG_DFLT;
boPin129Fault.ReceiverAdress :=1;
boPin129Fault.ToolScalingDivisor :=1;
boPin129Fault.ToolScalingMultiplier :=1;
boPin129Fault.ToolScalingOffset :=0;
boPin129Fault.ToolUnit :="";

boPin106Fault.AppScalingDivisor :=1;
boPin106Fault.AppScalingMultiplier :=1;
boPin106Fault.AppScalingOffset :=0;
boPin106Fault.AppUnit :="";
boPin106Fault.CanDefault :=0;
boPin106Fault.CanInit :=0;
boPin106Fault.CanMax :=1;
boPin106Fault.CanMin :=0;
boPin106Fault.CanUnit :="";
boPin106Fault.Description :="for the Neotec diag pages";
boPin106Fault.ErrorReaction := eErrorReaction.ERSIG_DFLT;
boPin106Fault.ReceiverAdress :=1;
boPin106Fault.ToolScalingDivisor :=1;
boPin106Fault.ToolScalingMultiplier :=1;
boPin106Fault.ToolScalingOffset :=0;
boPin106Fault.ToolUnit :="";

boPin130Fault.AppScalingDivisor :=1;
boPin130Fault.AppScalingMultiplier :=1;
boPin130Fault.AppScalingOffset :=0;
boPin130Fault.AppUnit :="";
boPin130Fault.CanDefault :=0;
boPin130Fault.CanInit :=0;
boPin130Fault.CanMax :=1;
boPin130Fault.CanMin :=0;
boPin130Fault.CanUnit :="";
boPin130Fault.Description :="for the Neotec diag pages";
boPin130Fault.ErrorReaction := eErrorReaction.ERSIG_DFLT;
boPin130Fault.ReceiverAdress :=1;
boPin130Fault.ToolScalingDivisor :=1;
boPin130Fault.ToolScalingMultiplier :=1;
boPin130Fault.ToolScalingOffset :=0;
boPin130Fault.ToolUnit :="";

boPin107Fault.AppScalingDivisor :=1;
boPin107Fault.AppScalingMultiplier :=1;
boPin107Fault.AppScalingOffset :=0;
boPin107Fault.AppUnit :="";
boPin107Fault.CanDefault :=0;
boPin107Fault.CanInit :=0;
boPin107Fault.CanMax :=1;
boPin107Fault.CanMin :=0;
boPin107Fault.CanUnit :="";
boPin107Fault.Description :="for the Neotec diag pages";
boPin107Fault.ErrorReaction := eErrorReaction.ERSIG_DFLT;
boPin107Fault.ReceiverAdress :=1;
boPin107Fault.ToolScalingDivisor :=1;
boPin107Fault.ToolScalingMultiplier :=1;
boPin107Fault.ToolScalingOffset :=0;
boPin107Fault.ToolUnit :="";

boPin131Fault.AppScalingDivisor :=1;
boPin131Fault.AppScalingMultiplier :=1;
boPin131Fault.AppScalingOffset :=0;
boPin131Fault.AppUnit :="";
boPin131Fault.CanDefault :=0;
boPin131Fault.CanInit :=0;
boPin131Fault.CanMax :=1;
boPin131Fault.CanMin :=0;
boPin131Fault.CanUnit :="";
boPin131Fault.Description :="for the Neotec diag pages";
boPin131Fault.ErrorReaction := eErrorReaction.ERSIG_DFLT;
boPin131Fault.ReceiverAdress :=1;
boPin131Fault.ToolScalingDivisor :=1;
boPin131Fault.ToolScalingMultiplier :=1;
boPin131Fault.ToolScalingOffset :=0;
boPin131Fault.ToolUnit :="";

boPin108Fault.AppScalingDivisor :=1;
boPin108Fault.AppScalingMultiplier :=1;
boPin108Fault.AppScalingOffset :=0;
boPin108Fault.AppUnit :="";
boPin108Fault.CanDefault :=0;
boPin108Fault.CanInit :=0;
boPin108Fault.CanMax :=1;
boPin108Fault.CanMin :=0;
boPin108Fault.CanUnit :="";
boPin108Fault.Description :="for the Neotec diag pages";
boPin108Fault.ErrorReaction := eErrorReaction.ERSIG_DFLT;
boPin108Fault.ReceiverAdress :=1;
boPin108Fault.ToolScalingDivisor :=1;
boPin108Fault.ToolScalingMultiplier :=1;
boPin108Fault.ToolScalingOffset :=0;
boPin108Fault.ToolUnit :="";

boPin132Fault.AppScalingDivisor :=1;
boPin132Fault.AppScalingMultiplier :=1;
boPin132Fault.AppScalingOffset :=0;
boPin132Fault.AppUnit :="";
boPin132Fault.CanDefault :=0;
boPin132Fault.CanInit :=0;
boPin132Fault.CanMax :=1;
boPin132Fault.CanMin :=0;
boPin132Fault.CanUnit :="";
boPin132Fault.Description :="for the Neotec diag pages";
boPin132Fault.ErrorReaction := eErrorReaction.ERSIG_DFLT;
boPin132Fault.ReceiverAdress :=1;
boPin132Fault.ToolScalingDivisor :=1;
boPin132Fault.ToolScalingMultiplier :=1;
boPin132Fault.ToolScalingOffset :=0;
boPin132Fault.ToolUnit :="";

boPin109Fault.AppScalingDivisor :=1;
boPin109Fault.AppScalingMultiplier :=1;
boPin109Fault.AppScalingOffset :=0;
boPin109Fault.AppUnit :="";
boPin109Fault.CanDefault :=0;
boPin109Fault.CanInit :=0;
boPin109Fault.CanMax :=1;
boPin109Fault.CanMin :=0;
boPin109Fault.CanUnit :="";
boPin109Fault.Description :="for the Neotec diag pages";
boPin109Fault.ErrorReaction := eErrorReaction.ERSIG_DFLT;
boPin109Fault.ReceiverAdress :=1;
boPin109Fault.ToolScalingDivisor :=1;
boPin109Fault.ToolScalingMultiplier :=1;
boPin109Fault.ToolScalingOffset :=0;
boPin109Fault.ToolUnit :="";

boPin133Fault.AppScalingDivisor :=1;
boPin133Fault.AppScalingMultiplier :=1;
boPin133Fault.AppScalingOffset :=0;
boPin133Fault.AppUnit :="";
boPin133Fault.CanDefault :=0;
boPin133Fault.CanInit :=0;
boPin133Fault.CanMax :=1;
boPin133Fault.CanMin :=0;
boPin133Fault.CanUnit :="";
boPin133Fault.Description :="for the Neotec diag pages";
boPin133Fault.ErrorReaction := eErrorReaction.ERSIG_DFLT;
boPin133Fault.ReceiverAdress :=1;
boPin133Fault.ToolScalingDivisor :=1;
boPin133Fault.ToolScalingMultiplier :=1;
boPin133Fault.ToolScalingOffset :=0;
boPin133Fault.ToolUnit :="";

boPin110Fault.AppScalingDivisor :=1;
boPin110Fault.AppScalingMultiplier :=1;
boPin110Fault.AppScalingOffset :=0;
boPin110Fault.AppUnit :="";
boPin110Fault.CanDefault :=0;
boPin110Fault.CanInit :=0;
boPin110Fault.CanMax :=1;
boPin110Fault.CanMin :=0;
boPin110Fault.CanUnit :="";
boPin110Fault.Description :="for the Neotec diag pages";
boPin110Fault.ErrorReaction := eErrorReaction.ERSIG_DFLT;
boPin110Fault.ReceiverAdress :=1;
boPin110Fault.ToolScalingDivisor :=1;
boPin110Fault.ToolScalingMultiplier :=1;
boPin110Fault.ToolScalingOffset :=0;
boPin110Fault.ToolUnit :="";

boPin134Fault.AppScalingDivisor :=1;
boPin134Fault.AppScalingMultiplier :=1;
boPin134Fault.AppScalingOffset :=0;
boPin134Fault.AppUnit :="";
boPin134Fault.CanDefault :=0;
boPin134Fault.CanInit :=0;
boPin134Fault.CanMax :=1;
boPin134Fault.CanMin :=0;
boPin134Fault.CanUnit :="";
boPin134Fault.Description :="for the Neotec diag pages";
boPin134Fault.ErrorReaction := eErrorReaction.ERSIG_DFLT;
boPin134Fault.ReceiverAdress :=1;
boPin134Fault.ToolScalingDivisor :=1;
boPin134Fault.ToolScalingMultiplier :=1;
boPin134Fault.ToolScalingOffset :=0;
boPin134Fault.ToolUnit :="";

boPin111Fault.AppScalingDivisor :=1;
boPin111Fault.AppScalingMultiplier :=1;
boPin111Fault.AppScalingOffset :=0;
boPin111Fault.AppUnit :="";
boPin111Fault.CanDefault :=0;
boPin111Fault.CanInit :=0;
boPin111Fault.CanMax :=1;
boPin111Fault.CanMin :=0;
boPin111Fault.CanUnit :="";
boPin111Fault.Description :="for the Neotec diag pages";
boPin111Fault.ErrorReaction := eErrorReaction.ERSIG_DFLT;
boPin111Fault.ReceiverAdress :=1;
boPin111Fault.ToolScalingDivisor :=1;
boPin111Fault.ToolScalingMultiplier :=1;
boPin111Fault.ToolScalingOffset :=0;
boPin111Fault.ToolUnit :="";

boPin135Fault.AppScalingDivisor :=1;
boPin135Fault.AppScalingMultiplier :=1;
boPin135Fault.AppScalingOffset :=0;
boPin135Fault.AppUnit :="";
boPin135Fault.CanDefault :=0;
boPin135Fault.CanInit :=0;
boPin135Fault.CanMax :=1;
boPin135Fault.CanMin :=0;
boPin135Fault.CanUnit :="";
boPin135Fault.Description :="for the Neotec diag pages";
boPin135Fault.ErrorReaction := eErrorReaction.ERSIG_DFLT;
boPin135Fault.ReceiverAdress :=1;
boPin135Fault.ToolScalingDivisor :=1;
boPin135Fault.ToolScalingMultiplier :=1;
boPin135Fault.ToolScalingOffset :=0;
boPin135Fault.ToolUnit :="";

boPin112Fault.AppScalingDivisor :=1;
boPin112Fault.AppScalingMultiplier :=1;
boPin112Fault.AppScalingOffset :=0;
boPin112Fault.AppUnit :="";
boPin112Fault.CanDefault :=0;
boPin112Fault.CanInit :=0;
boPin112Fault.CanMax :=1;
boPin112Fault.CanMin :=0;
boPin112Fault.CanUnit :="";
boPin112Fault.Description :="for the Neotec diag pages";
boPin112Fault.ErrorReaction := eErrorReaction.ERSIG_DFLT;
boPin112Fault.ReceiverAdress :=1;
boPin112Fault.ToolScalingDivisor :=1;
boPin112Fault.ToolScalingMultiplier :=1;
boPin112Fault.ToolScalingOffset :=0;
boPin112Fault.ToolUnit :="";

boPin136Fault.AppScalingDivisor :=1;
boPin136Fault.AppScalingMultiplier :=1;
boPin136Fault.AppScalingOffset :=0;
boPin136Fault.AppUnit :="";
boPin136Fault.CanDefault :=0;
boPin136Fault.CanInit :=0;
boPin136Fault.CanMax :=1;
boPin136Fault.CanMin :=0;
boPin136Fault.CanUnit :="";
boPin136Fault.Description :="for the Neotec diag pages";
boPin136Fault.ErrorReaction := eErrorReaction.ERSIG_DFLT;
boPin136Fault.ReceiverAdress :=1;
boPin136Fault.ToolScalingDivisor :=1;
boPin136Fault.ToolScalingMultiplier :=1;
boPin136Fault.ToolScalingOffset :=0;
boPin136Fault.ToolUnit :="";

boPin113Fault.AppScalingDivisor :=1;
boPin113Fault.AppScalingMultiplier :=1;
boPin113Fault.AppScalingOffset :=0;
boPin113Fault.AppUnit :="";
boPin113Fault.CanDefault :=0;
boPin113Fault.CanInit :=0;
boPin113Fault.CanMax :=1;
boPin113Fault.CanMin :=0;
boPin113Fault.CanUnit :="";
boPin113Fault.Description :="for the Neotec diag pages";
boPin113Fault.ErrorReaction := eErrorReaction.ERSIG_DFLT;
boPin113Fault.ReceiverAdress :=1;
boPin113Fault.ToolScalingDivisor :=1;
boPin113Fault.ToolScalingMultiplier :=1;
boPin113Fault.ToolScalingOffset :=0;
boPin113Fault.ToolUnit :="";

boPin137Fault.AppScalingDivisor :=1;
boPin137Fault.AppScalingMultiplier :=1;
boPin137Fault.AppScalingOffset :=0;
boPin137Fault.AppUnit :="";
boPin137Fault.CanDefault :=0;
boPin137Fault.CanInit :=0;
boPin137Fault.CanMax :=1;
boPin137Fault.CanMin :=0;
boPin137Fault.CanUnit :="";
boPin137Fault.Description :="for the Neotec diag pages";
boPin137Fault.ErrorReaction := eErrorReaction.ERSIG_DFLT;
boPin137Fault.ReceiverAdress :=1;
boPin137Fault.ToolScalingDivisor :=1;
boPin137Fault.ToolScalingMultiplier :=1;
boPin137Fault.ToolScalingOffset :=0;
boPin137Fault.ToolUnit :="";

boPin114Fault.AppScalingDivisor :=1;
boPin114Fault.AppScalingMultiplier :=1;
boPin114Fault.AppScalingOffset :=0;
boPin114Fault.AppUnit :="";
boPin114Fault.CanDefault :=0;
boPin114Fault.CanInit :=0;
boPin114Fault.CanMax :=1;
boPin114Fault.CanMin :=0;
boPin114Fault.CanUnit :="";
boPin114Fault.Description :="for the Neotec diag pages";
boPin114Fault.ErrorReaction := eErrorReaction.ERSIG_DFLT;
boPin114Fault.ReceiverAdress :=1;
boPin114Fault.ToolScalingDivisor :=1;
boPin114Fault.ToolScalingMultiplier :=1;
boPin114Fault.ToolScalingOffset :=0;
boPin114Fault.ToolUnit :="";

boPin138Fault.AppScalingDivisor :=1;
boPin138Fault.AppScalingMultiplier :=1;
boPin138Fault.AppScalingOffset :=0;
boPin138Fault.AppUnit :="";
boPin138Fault.CanDefault :=0;
boPin138Fault.CanInit :=0;
boPin138Fault.CanMax :=1;
boPin138Fault.CanMin :=0;
boPin138Fault.CanUnit :="";
boPin138Fault.Description :="for the Neotec diag pages";
boPin138Fault.ErrorReaction := eErrorReaction.ERSIG_DFLT;
boPin138Fault.ReceiverAdress :=1;
boPin138Fault.ToolScalingDivisor :=1;
boPin138Fault.ToolScalingMultiplier :=1;
boPin138Fault.ToolScalingOffset :=0;
boPin138Fault.ToolUnit :="";

boPin115Fault.AppScalingDivisor :=1;
boPin115Fault.AppScalingMultiplier :=1;
boPin115Fault.AppScalingOffset :=0;
boPin115Fault.AppUnit :="";
boPin115Fault.CanDefault :=0;
boPin115Fault.CanInit :=0;
boPin115Fault.CanMax :=1;
boPin115Fault.CanMin :=0;
boPin115Fault.CanUnit :="";
boPin115Fault.Description :="for the Neotec diag pages";
boPin115Fault.ErrorReaction := eErrorReaction.ERSIG_DFLT;
boPin115Fault.ReceiverAdress :=1;
boPin115Fault.ToolScalingDivisor :=1;
boPin115Fault.ToolScalingMultiplier :=1;
boPin115Fault.ToolScalingOffset :=0;
boPin115Fault.ToolUnit :="";

boPin139Fault.AppScalingDivisor :=1;
boPin139Fault.AppScalingMultiplier :=1;
boPin139Fault.AppScalingOffset :=0;
boPin139Fault.AppUnit :="";
boPin139Fault.CanDefault :=0;
boPin139Fault.CanInit :=0;
boPin139Fault.CanMax :=1;
boPin139Fault.CanMin :=0;
boPin139Fault.CanUnit :="";
boPin139Fault.Description :="for the Neotec diag pages";
boPin139Fault.ErrorReaction := eErrorReaction.ERSIG_DFLT;
boPin139Fault.ReceiverAdress :=1;
boPin139Fault.ToolScalingDivisor :=1;
boPin139Fault.ToolScalingMultiplier :=1;
boPin139Fault.ToolScalingOffset :=0;
boPin139Fault.ToolUnit :="";

boPin116Fault.AppScalingDivisor :=1;
boPin116Fault.AppScalingMultiplier :=1;
boPin116Fault.AppScalingOffset :=0;
boPin116Fault.AppUnit :="";
boPin116Fault.CanDefault :=0;
boPin116Fault.CanInit :=0;
boPin116Fault.CanMax :=1;
boPin116Fault.CanMin :=0;
boPin116Fault.CanUnit :="";
boPin116Fault.Description :="for the Neotec diag pages";
boPin116Fault.ErrorReaction := eErrorReaction.ERSIG_DFLT;
boPin116Fault.ReceiverAdress :=1;
boPin116Fault.ToolScalingDivisor :=1;
boPin116Fault.ToolScalingMultiplier :=1;
boPin116Fault.ToolScalingOffset :=0;
boPin116Fault.ToolUnit :="";

boPin140Fault.AppScalingDivisor :=1;
boPin140Fault.AppScalingMultiplier :=1;
boPin140Fault.AppScalingOffset :=0;
boPin140Fault.AppUnit :="";
boPin140Fault.CanDefault :=0;
boPin140Fault.CanInit :=0;
boPin140Fault.CanMax :=1;
boPin140Fault.CanMin :=0;
boPin140Fault.CanUnit :="";
boPin140Fault.Description :="for the Neotec diag pages";
boPin140Fault.ErrorReaction := eErrorReaction.ERSIG_DFLT;
boPin140Fault.ReceiverAdress :=1;
boPin140Fault.ToolScalingDivisor :=1;
boPin140Fault.ToolScalingMultiplier :=1;
boPin140Fault.ToolScalingOffset :=0;
boPin140Fault.ToolUnit :="";

boPin117Fault.AppScalingDivisor :=1;
boPin117Fault.AppScalingMultiplier :=1;
boPin117Fault.AppScalingOffset :=0;
boPin117Fault.AppUnit :="";
boPin117Fault.CanDefault :=0;
boPin117Fault.CanInit :=0;
boPin117Fault.CanMax :=1;
boPin117Fault.CanMin :=0;
boPin117Fault.CanUnit :="";
boPin117Fault.Description :="for the Neotec diag pages";
boPin117Fault.ErrorReaction := eErrorReaction.ERSIG_DFLT;
boPin117Fault.ReceiverAdress :=1;
boPin117Fault.ToolScalingDivisor :=1;
boPin117Fault.ToolScalingMultiplier :=1;
boPin117Fault.ToolScalingOffset :=0;
boPin117Fault.ToolUnit :="";

boPin141Fault.AppScalingDivisor :=1;
boPin141Fault.AppScalingMultiplier :=1;
boPin141Fault.AppScalingOffset :=0;
boPin141Fault.AppUnit :="";
boPin141Fault.CanDefault :=0;
boPin141Fault.CanInit :=0;
boPin141Fault.CanMax :=1;
boPin141Fault.CanMin :=0;
boPin141Fault.CanUnit :="";
boPin141Fault.Description :="for the Neotec diag pages";
boPin141Fault.ErrorReaction := eErrorReaction.ERSIG_DFLT;
boPin141Fault.ReceiverAdress :=1;
boPin141Fault.ToolScalingDivisor :=1;
boPin141Fault.ToolScalingMultiplier :=1;
boPin141Fault.ToolScalingOffset :=0;
boPin141Fault.ToolUnit :="";

boPin122Fault.AppScalingDivisor :=1;
boPin122Fault.AppScalingMultiplier :=1;
boPin122Fault.AppScalingOffset :=0;
boPin122Fault.AppUnit :="";
boPin122Fault.CanDefault :=0;
boPin122Fault.CanInit :=0;
boPin122Fault.CanMax :=1;
boPin122Fault.CanMin :=0;
boPin122Fault.CanUnit :="";
boPin122Fault.Description :="for the Neotec diag pages";
boPin122Fault.ErrorReaction := eErrorReaction.ERSIG_DFLT;
boPin122Fault.ReceiverAdress :=1;
boPin122Fault.ToolScalingDivisor :=1;
boPin122Fault.ToolScalingMultiplier :=1;
boPin122Fault.ToolScalingOffset :=0;
boPin122Fault.ToolUnit :="";

boPin146Fault.AppScalingDivisor :=1;
boPin146Fault.AppScalingMultiplier :=1;
boPin146Fault.AppScalingOffset :=0;
boPin146Fault.AppUnit :="";
boPin146Fault.CanDefault :=0;
boPin146Fault.CanInit :=0;
boPin146Fault.CanMax :=1;
boPin146Fault.CanMin :=0;
boPin146Fault.CanUnit :="";
boPin146Fault.Description :="for the Neotec diag pages";
boPin146Fault.ErrorReaction := eErrorReaction.ERSIG_DFLT;
boPin146Fault.ReceiverAdress :=1;
boPin146Fault.ToolScalingDivisor :=1;
boPin146Fault.ToolScalingMultiplier :=1;
boPin146Fault.ToolScalingOffset :=0;
boPin146Fault.ToolUnit :="";

boPin123Fault.AppScalingDivisor :=1;
boPin123Fault.AppScalingMultiplier :=1;
boPin123Fault.AppScalingOffset :=0;
boPin123Fault.AppUnit :="";
boPin123Fault.CanDefault :=0;
boPin123Fault.CanInit :=0;
boPin123Fault.CanMax :=1;
boPin123Fault.CanMin :=0;
boPin123Fault.CanUnit :="";
boPin123Fault.Description :="for the Neotec diag pages";
boPin123Fault.ErrorReaction := eErrorReaction.ERSIG_DFLT;
boPin123Fault.ReceiverAdress :=1;
boPin123Fault.ToolScalingDivisor :=1;
boPin123Fault.ToolScalingMultiplier :=1;
boPin123Fault.ToolScalingOffset :=0;
boPin123Fault.ToolUnit :="";

boPin147Fault.AppScalingDivisor :=1;
boPin147Fault.AppScalingMultiplier :=1;
boPin147Fault.AppScalingOffset :=0;
boPin147Fault.AppUnit :="";
boPin147Fault.CanDefault :=0;
boPin147Fault.CanInit :=0;
boPin147Fault.CanMax :=1;
boPin147Fault.CanMin :=0;
boPin147Fault.CanUnit :="";
boPin147Fault.Description :="for the Neotec diag pages";
boPin147Fault.ErrorReaction := eErrorReaction.ERSIG_DFLT;
boPin147Fault.ReceiverAdress :=1;
boPin147Fault.ToolScalingDivisor :=1;
boPin147Fault.ToolScalingMultiplier :=1;
boPin147Fault.ToolScalingOffset :=0;
boPin147Fault.ToolUnit :="";

boPin124Fault.AppScalingDivisor :=1;
boPin124Fault.AppScalingMultiplier :=1;
boPin124Fault.AppScalingOffset :=0;
boPin124Fault.AppUnit :="";
boPin124Fault.CanDefault :=0;
boPin124Fault.CanInit :=0;
boPin124Fault.CanMax :=1;
boPin124Fault.CanMin :=0;
boPin124Fault.CanUnit :="";
boPin124Fault.Description :="for the Neotec diag pages";
boPin124Fault.ErrorReaction := eErrorReaction.ERSIG_DFLT;
boPin124Fault.ReceiverAdress :=1;
boPin124Fault.ToolScalingDivisor :=1;
boPin124Fault.ToolScalingMultiplier :=1;
boPin124Fault.ToolScalingOffset :=0;
boPin124Fault.ToolUnit :="";

boPin148Fault.AppScalingDivisor :=1;
boPin148Fault.AppScalingMultiplier :=1;
boPin148Fault.AppScalingOffset :=0;
boPin148Fault.AppUnit :="";
boPin148Fault.CanDefault :=0;
boPin148Fault.CanInit :=0;
boPin148Fault.CanMax :=1;
boPin148Fault.CanMin :=0;
boPin148Fault.CanUnit :="";
boPin148Fault.Description :="for the Neotec diag pages";
boPin148Fault.ErrorReaction := eErrorReaction.ERSIG_DFLT;
boPin148Fault.ReceiverAdress :=1;
boPin148Fault.ToolScalingDivisor :=1;
boPin148Fault.ToolScalingMultiplier :=1;
boPin148Fault.ToolScalingOffset :=0;
boPin148Fault.ToolUnit :="";

boPin153Fault.AppScalingDivisor :=1;
boPin153Fault.AppScalingMultiplier :=1;
boPin153Fault.AppScalingOffset :=0;
boPin153Fault.AppUnit :="";
boPin153Fault.CanDefault :=0;
boPin153Fault.CanInit :=0;
boPin153Fault.CanMax :=1;
boPin153Fault.CanMin :=0;
boPin153Fault.CanUnit :="";
boPin153Fault.Description :="for the Neotec diag pages";
boPin153Fault.ErrorReaction := eErrorReaction.ERSIG_DFLT;
boPin153Fault.ReceiverAdress :=1;
boPin153Fault.ToolScalingDivisor :=1;
boPin153Fault.ToolScalingMultiplier :=1;
boPin153Fault.ToolScalingOffset :=0;
boPin153Fault.ToolUnit :="";

boPin177Fault.AppScalingDivisor :=1;
boPin177Fault.AppScalingMultiplier :=1;
boPin177Fault.AppScalingOffset :=0;
boPin177Fault.AppUnit :="";
boPin177Fault.CanDefault :=0;
boPin177Fault.CanInit :=0;
boPin177Fault.CanMax :=1;
boPin177Fault.CanMin :=0;
boPin177Fault.CanUnit :="";
boPin177Fault.Description :="for the Neotec diag pages";
boPin177Fault.ErrorReaction := eErrorReaction.ERSIG_DFLT;
boPin177Fault.ReceiverAdress :=1;
boPin177Fault.ToolScalingDivisor :=1;
boPin177Fault.ToolScalingMultiplier :=1;
boPin177Fault.ToolScalingOffset :=0;
boPin177Fault.ToolUnit :="";

boPin156Fault.AppScalingDivisor :=1;
boPin156Fault.AppScalingMultiplier :=1;
boPin156Fault.AppScalingOffset :=0;
boPin156Fault.AppUnit :="";
boPin156Fault.CanDefault :=0;
boPin156Fault.CanInit :=0;
boPin156Fault.CanMax :=1;
boPin156Fault.CanMin :=0;
boPin156Fault.CanUnit :="";
boPin156Fault.Description :="for the Neotec diag pages";
boPin156Fault.ErrorReaction := eErrorReaction.ERSIG_DFLT;
boPin156Fault.ReceiverAdress :=1;
boPin156Fault.ToolScalingDivisor :=1;
boPin156Fault.ToolScalingMultiplier :=1;
boPin156Fault.ToolScalingOffset :=0;
boPin156Fault.ToolUnit :="";

boPin180Fault.AppScalingDivisor :=1;
boPin180Fault.AppScalingMultiplier :=1;
boPin180Fault.AppScalingOffset :=0;
boPin180Fault.AppUnit :="";
boPin180Fault.CanDefault :=0;
boPin180Fault.CanInit :=0;
boPin180Fault.CanMax :=1;
boPin180Fault.CanMin :=0;
boPin180Fault.CanUnit :="";
boPin180Fault.Description :="for the Neotec diag pages";
boPin180Fault.ErrorReaction := eErrorReaction.ERSIG_DFLT;
boPin180Fault.ReceiverAdress :=1;
boPin180Fault.ToolScalingDivisor :=1;
boPin180Fault.ToolScalingMultiplier :=1;
boPin180Fault.ToolScalingOffset :=0;
boPin180Fault.ToolUnit :="";

boPin159Fault.AppScalingDivisor :=1;
boPin159Fault.AppScalingMultiplier :=1;
boPin159Fault.AppScalingOffset :=0;
boPin159Fault.AppUnit :="";
boPin159Fault.CanDefault :=0;
boPin159Fault.CanInit :=0;
boPin159Fault.CanMax :=1;
boPin159Fault.CanMin :=0;
boPin159Fault.CanUnit :="";
boPin159Fault.Description :="for the Neotec diag pages";
boPin159Fault.ErrorReaction := eErrorReaction.ERSIG_DFLT;
boPin159Fault.ReceiverAdress :=1;
boPin159Fault.ToolScalingDivisor :=1;
boPin159Fault.ToolScalingMultiplier :=1;
boPin159Fault.ToolScalingOffset :=0;
boPin159Fault.ToolUnit :="";

boPin183Fault.AppScalingDivisor :=1;
boPin183Fault.AppScalingMultiplier :=1;
boPin183Fault.AppScalingOffset :=0;
boPin183Fault.AppUnit :="";
boPin183Fault.CanDefault :=0;
boPin183Fault.CanInit :=0;
boPin183Fault.CanMax :=1;
boPin183Fault.CanMin :=0;
boPin183Fault.CanUnit :="";
boPin183Fault.Description :="for the Neotec diag pages";
boPin183Fault.ErrorReaction := eErrorReaction.ERSIG_DFLT;
boPin183Fault.ReceiverAdress :=1;
boPin183Fault.ToolScalingDivisor :=1;
boPin183Fault.ToolScalingMultiplier :=1;
boPin183Fault.ToolScalingOffset :=0;
boPin183Fault.ToolUnit :="";

boPin186Fault.AppScalingDivisor :=1;
boPin186Fault.AppScalingMultiplier :=1;
boPin186Fault.AppScalingOffset :=0;
boPin186Fault.AppUnit :="";
boPin186Fault.CanDefault :=0;
boPin186Fault.CanInit :=0;
boPin186Fault.CanMax :=1;
boPin186Fault.CanMin :=0;
boPin186Fault.CanUnit :="";
boPin186Fault.Description :="for the Neotec diag pages";
boPin186Fault.ErrorReaction := eErrorReaction.ERSIG_DFLT;
boPin186Fault.ReceiverAdress :=1;
boPin186Fault.ToolScalingDivisor :=1;
boPin186Fault.ToolScalingMultiplier :=1;
boPin186Fault.ToolScalingOffset :=0;
boPin186Fault.ToolUnit :="";

boPin162Fault.AppScalingDivisor :=1;
boPin162Fault.AppScalingMultiplier :=1;
boPin162Fault.AppScalingOffset :=0;
boPin162Fault.AppUnit :="";
boPin162Fault.CanDefault :=0;
boPin162Fault.CanInit :=0;
boPin162Fault.CanMax :=1;
boPin162Fault.CanMin :=0;
boPin162Fault.CanUnit :="";
boPin162Fault.Description :="for the Neotec diag pages";
boPin162Fault.ErrorReaction := eErrorReaction.ERSIG_DFLT;
boPin162Fault.ReceiverAdress :=1;
boPin162Fault.ToolScalingDivisor :=1;
boPin162Fault.ToolScalingMultiplier :=1;
boPin162Fault.ToolScalingOffset :=0;
boPin162Fault.ToolUnit :="";

boPin189Fault.AppScalingDivisor :=1;
boPin189Fault.AppScalingMultiplier :=1;
boPin189Fault.AppScalingOffset :=0;
boPin189Fault.AppUnit :="";
boPin189Fault.CanDefault :=0;
boPin189Fault.CanInit :=0;
boPin189Fault.CanMax :=1;
boPin189Fault.CanMin :=0;
boPin189Fault.CanUnit :="";
boPin189Fault.Description :="for the Neotec diag pages";
boPin189Fault.ErrorReaction := eErrorReaction.ERSIG_DFLT;
boPin189Fault.ReceiverAdress :=1;
boPin189Fault.ToolScalingDivisor :=1;
boPin189Fault.ToolScalingMultiplier :=1;
boPin189Fault.ToolScalingOffset :=0;
boPin189Fault.ToolUnit :="";

boPin165Fault.AppScalingDivisor :=1;
boPin165Fault.AppScalingMultiplier :=1;
boPin165Fault.AppScalingOffset :=0;
boPin165Fault.AppUnit :="";
boPin165Fault.CanDefault :=0;
boPin165Fault.CanInit :=0;
boPin165Fault.CanMax :=1;
boPin165Fault.CanMin :=0;
boPin165Fault.CanUnit :="";
boPin165Fault.Description :="for the Neotec diag pages";
boPin165Fault.ErrorReaction := eErrorReaction.ERSIG_DFLT;
boPin165Fault.ReceiverAdress :=1;
boPin165Fault.ToolScalingDivisor :=1;
boPin165Fault.ToolScalingMultiplier :=1;
boPin165Fault.ToolScalingOffset :=0;
boPin165Fault.ToolUnit :="";

boPin192Fault.AppScalingDivisor :=1;
boPin192Fault.AppScalingMultiplier :=1;
boPin192Fault.AppScalingOffset :=0;
boPin192Fault.AppUnit :="";
boPin192Fault.CanDefault :=0;
boPin192Fault.CanInit :=0;
boPin192Fault.CanMax :=1;
boPin192Fault.CanMin :=0;
boPin192Fault.CanUnit :="";
boPin192Fault.Description :="for the Neotec diag pages";
boPin192Fault.ErrorReaction := eErrorReaction.ERSIG_DFLT;
boPin192Fault.ReceiverAdress :=1;
boPin192Fault.ToolScalingDivisor :=1;
boPin192Fault.ToolScalingMultiplier :=1;
boPin192Fault.ToolScalingOffset :=0;
boPin192Fault.ToolUnit :="";

boPin168Fault.AppScalingDivisor :=1;
boPin168Fault.AppScalingMultiplier :=1;
boPin168Fault.AppScalingOffset :=0;
boPin168Fault.AppUnit :="";
boPin168Fault.CanDefault :=0;
boPin168Fault.CanInit :=0;
boPin168Fault.CanMax :=1;
boPin168Fault.CanMin :=0;
boPin168Fault.CanUnit :="";
boPin168Fault.Description :="for the Neotec diag pages";
boPin168Fault.ErrorReaction := eErrorReaction.ERSIG_DFLT;
boPin168Fault.ReceiverAdress :=1;
boPin168Fault.ToolScalingDivisor :=1;
boPin168Fault.ToolScalingMultiplier :=1;
boPin168Fault.ToolScalingOffset :=0;
boPin168Fault.ToolUnit :="";

boPin195Fault.AppScalingDivisor :=1;
boPin195Fault.AppScalingMultiplier :=1;
boPin195Fault.AppScalingOffset :=0;
boPin195Fault.AppUnit :="";
boPin195Fault.CanDefault :=0;
boPin195Fault.CanInit :=0;
boPin195Fault.CanMax :=1;
boPin195Fault.CanMin :=0;
boPin195Fault.CanUnit :="";
boPin195Fault.Description :="for the Neotec diag pages";
boPin195Fault.ErrorReaction := eErrorReaction.ERSIG_DFLT;
boPin195Fault.ReceiverAdress :=1;
boPin195Fault.ToolScalingDivisor :=1;
boPin195Fault.ToolScalingMultiplier :=1;
boPin195Fault.ToolScalingOffset :=0;
boPin195Fault.ToolUnit :="";

boPin171Fault.AppScalingDivisor :=1;
boPin171Fault.AppScalingMultiplier :=1;
boPin171Fault.AppScalingOffset :=0;
boPin171Fault.AppUnit :="";
boPin171Fault.CanDefault :=0;
boPin171Fault.CanInit :=0;
boPin171Fault.CanMax :=1;
boPin171Fault.CanMin :=0;
boPin171Fault.CanUnit :="";
boPin171Fault.Description :="for the Neotec diag pages";
boPin171Fault.ErrorReaction := eErrorReaction.ERSIG_DFLT;
boPin171Fault.ReceiverAdress :=1;
boPin171Fault.ToolScalingDivisor :=1;
boPin171Fault.ToolScalingMultiplier :=1;
boPin171Fault.ToolScalingOffset :=0;
boPin171Fault.ToolUnit :="";

boPin154Fault.AppScalingDivisor :=1;
boPin154Fault.AppScalingMultiplier :=1;
boPin154Fault.AppScalingOffset :=0;
boPin154Fault.AppUnit :="";
boPin154Fault.CanDefault :=0;
boPin154Fault.CanInit :=0;
boPin154Fault.CanMax :=1;
boPin154Fault.CanMin :=0;
boPin154Fault.CanUnit :="";
boPin154Fault.Description :="for the Neotec diag pages";
boPin154Fault.ErrorReaction := eErrorReaction.ERSIG_DFLT;
boPin154Fault.ReceiverAdress :=1;
boPin154Fault.ToolScalingDivisor :=1;
boPin154Fault.ToolScalingMultiplier :=1;
boPin154Fault.ToolScalingOffset :=0;
boPin154Fault.ToolUnit :="";

boPin178Fault.AppScalingDivisor :=1;
boPin178Fault.AppScalingMultiplier :=1;
boPin178Fault.AppScalingOffset :=0;
boPin178Fault.AppUnit :="";
boPin178Fault.CanDefault :=0;
boPin178Fault.CanInit :=0;
boPin178Fault.CanMax :=1;
boPin178Fault.CanMin :=0;
boPin178Fault.CanUnit :="";
boPin178Fault.Description :="for the Neotec diag pages";
boPin178Fault.ErrorReaction := eErrorReaction.ERSIG_DFLT;
boPin178Fault.ReceiverAdress :=1;
boPin178Fault.ToolScalingDivisor :=1;
boPin178Fault.ToolScalingMultiplier :=1;
boPin178Fault.ToolScalingOffset :=0;
boPin178Fault.ToolUnit :="";

boPin157Fault.AppScalingDivisor :=1;
boPin157Fault.AppScalingMultiplier :=1;
boPin157Fault.AppScalingOffset :=0;
boPin157Fault.AppUnit :="";
boPin157Fault.CanDefault :=0;
boPin157Fault.CanInit :=0;
boPin157Fault.CanMax :=1;
boPin157Fault.CanMin :=0;
boPin157Fault.CanUnit :="";
boPin157Fault.Description :="for the Neotec diag pages";
boPin157Fault.ErrorReaction := eErrorReaction.ERSIG_DFLT;
boPin157Fault.ReceiverAdress :=1;
boPin157Fault.ToolScalingDivisor :=1;
boPin157Fault.ToolScalingMultiplier :=1;
boPin157Fault.ToolScalingOffset :=0;
boPin157Fault.ToolUnit :="";


                
END_METHOD
END_FUNCTION_BLOCK

FUNCTION_BLOCK Msg6C0SendToEvision7MessageClass EXTENDS CanReceiveMessageClass
  VAR_INPUT
    boPin181Fault : BoolCanSignalClass;
    boPin160Fault : BoolCanSignalClass;
    boPin184Fault : BoolCanSignalClass;
    boPin187Fault : BoolCanSignalClass;
    boPin163Fault : BoolCanSignalClass;
    boPin190Fault : BoolCanSignalClass;
    boPin166Fault : BoolCanSignalClass;
    boPin193Fault : BoolCanSignalClass;
    boPin169Fault : BoolCanSignalClass;
    boPin196Fault : BoolCanSignalClass;
    boPin172Fault : BoolCanSignalClass;
    boPin101Fault : BoolCanSignalClass;
    boPin125Fault : BoolCanSignalClass;
    boPin150Fault : BoolCanSignalClass;
    boPin174Fault : BoolCanSignalClass;
    boPin102Fault : BoolCanSignalClass;
    boPin126Fault : BoolCanSignalClass;
    boPin151Fault : BoolCanSignalClass;
    boPin175Fault : BoolCanSignalClass;
    boPin149Fault : BoolCanSignalClass;
    boPin173Fault : BoolCanSignalClass;
    boPin152Fault : BoolCanSignalClass;
    boPin176Fault : BoolCanSignalClass;
    boPin155Fault : BoolCanSignalClass;
    boPin179Fault : BoolCanSignalClass;
    boPin158Fault : BoolCanSignalClass;
    boPin182Fault : BoolCanSignalClass;
    boPin251Fault : BoolCanSignalClass;
    boPin238Fault : BoolCanSignalClass;
    boPin252Fault : BoolCanSignalClass;
    boPin239Fault : BoolCanSignalClass;
    boPin253Fault : BoolCanSignalClass;
    boPin240Fault : BoolCanSignalClass;
    boPin254Fault : BoolCanSignalClass;
    boPin241Fault : BoolCanSignalClass;
    boPin161Fault : BoolCanSignalClass;
    boPin185Fault : BoolCanSignalClass;
    boPin188Fault : BoolCanSignalClass;
    boPin164Fault : BoolCanSignalClass;
    boPin191Fault : BoolCanSignalClass;
    boPin167Fault : BoolCanSignalClass;
    boPin194Fault : BoolCanSignalClass;
    boPin170Fault : BoolCanSignalClass;
    Counter : UInt32CanSignalClass;
  END_VAR

            
          

METHOD SetData
  VAR_INPUT
    CanMsgPointer : POINTER TO CanMessageClass;
  END_VAR
                  IF IsValidPointer(canMsgPointer,'SetData') THEN
	SUPER^.SetData(CanMsgPointer);
	//Set the new data
	boPin181Fault.Value := canMsgPointer^.GetBoolOnBit(0);
	boPin160Fault.Value := canMsgPointer^.GetBoolOnBit(1);
	boPin184Fault.Value := canMsgPointer^.GetBoolOnBit(2);
	boPin187Fault.Value := canMsgPointer^.GetBoolOnBit(3);
	boPin163Fault.Value := canMsgPointer^.GetBoolOnBit(4);
	boPin190Fault.Value := canMsgPointer^.GetBoolOnBit(5);
	boPin166Fault.Value := canMsgPointer^.GetBoolOnBit(6);
	boPin193Fault.Value := canMsgPointer^.GetBoolOnBit(7);
	boPin169Fault.Value := canMsgPointer^.GetBoolOnBit(8);
	boPin196Fault.Value := canMsgPointer^.GetBoolOnBit(9);
	boPin172Fault.Value := canMsgPointer^.GetBoolOnBit(10);
	boPin101Fault.Value := canMsgPointer^.GetBoolOnBit(11);
	boPin125Fault.Value := canMsgPointer^.GetBoolOnBit(12);
	boPin150Fault.Value := canMsgPointer^.GetBoolOnBit(13);
	boPin174Fault.Value := canMsgPointer^.GetBoolOnBit(14);
	boPin102Fault.Value := canMsgPointer^.GetBoolOnBit(15);
	boPin126Fault.Value := canMsgPointer^.GetBoolOnBit(16);
	boPin151Fault.Value := canMsgPointer^.GetBoolOnBit(17);
	boPin175Fault.Value := canMsgPointer^.GetBoolOnBit(18);
	boPin149Fault.Value := canMsgPointer^.GetBoolOnBit(19);
	boPin173Fault.Value := canMsgPointer^.GetBoolOnBit(20);
	boPin152Fault.Value := canMsgPointer^.GetBoolOnBit(21);
	boPin176Fault.Value := canMsgPointer^.GetBoolOnBit(22);
	boPin155Fault.Value := canMsgPointer^.GetBoolOnBit(23);
	boPin179Fault.Value := canMsgPointer^.GetBoolOnBit(24);
	boPin158Fault.Value := canMsgPointer^.GetBoolOnBit(25);
	boPin182Fault.Value := canMsgPointer^.GetBoolOnBit(26);
	boPin251Fault.Value := canMsgPointer^.GetBoolOnBit(27);
	boPin238Fault.Value := canMsgPointer^.GetBoolOnBit(28);
	boPin252Fault.Value := canMsgPointer^.GetBoolOnBit(29);
	boPin239Fault.Value := canMsgPointer^.GetBoolOnBit(30);
	boPin253Fault.Value := canMsgPointer^.GetBoolOnBit(31);
	boPin240Fault.Value := canMsgPointer^.GetBoolOnBit(32);
	boPin254Fault.Value := canMsgPointer^.GetBoolOnBit(33);
	boPin241Fault.Value := canMsgPointer^.GetBoolOnBit(34);
	boPin161Fault.Value := canMsgPointer^.GetBoolOnBit(35);
	boPin185Fault.Value := canMsgPointer^.GetBoolOnBit(36);
	boPin188Fault.Value := canMsgPointer^.GetBoolOnBit(37);
	boPin164Fault.Value := canMsgPointer^.GetBoolOnBit(38);
	boPin191Fault.Value := canMsgPointer^.GetBoolOnBit(39);
	boPin167Fault.Value := canMsgPointer^.GetBoolOnBit(40);
	boPin194Fault.Value := canMsgPointer^.GetBoolOnBit(41);
	boPin170Fault.Value := canMsgPointer^.GetBoolOnBit(42);
	//And increase the counter
	Counter.Value := CanMsgPointer^.Counter.Value;
END_IF

                
END_METHOD

PROPERTY boPin181FaultRawValue : BOOL
GET
                    boPin181FaultRawValue := boPin181Fault.Value;

                  
END_GET
END_PROPERTY

PROPERTY boPin160FaultRawValue : BOOL
GET
                    boPin160FaultRawValue := boPin160Fault.Value;

                  
END_GET
END_PROPERTY

PROPERTY boPin184FaultRawValue : BOOL
GET
                    boPin184FaultRawValue := boPin184Fault.Value;

                  
END_GET
END_PROPERTY

PROPERTY boPin187FaultRawValue : BOOL
GET
                    boPin187FaultRawValue := boPin187Fault.Value;

                  
END_GET
END_PROPERTY

PROPERTY boPin163FaultRawValue : BOOL
GET
                    boPin163FaultRawValue := boPin163Fault.Value;

                  
END_GET
END_PROPERTY

PROPERTY boPin190FaultRawValue : BOOL
GET
                    boPin190FaultRawValue := boPin190Fault.Value;

                  
END_GET
END_PROPERTY

PROPERTY boPin166FaultRawValue : BOOL
GET
                    boPin166FaultRawValue := boPin166Fault.Value;

                  
END_GET
END_PROPERTY

PROPERTY boPin193FaultRawValue : BOOL
GET
                    boPin193FaultRawValue := boPin193Fault.Value;

                  
END_GET
END_PROPERTY

PROPERTY boPin169FaultRawValue : BOOL
GET
                    boPin169FaultRawValue := boPin169Fault.Value;

                  
END_GET
END_PROPERTY

PROPERTY boPin196FaultRawValue : BOOL
GET
                    boPin196FaultRawValue := boPin196Fault.Value;

                  
END_GET
END_PROPERTY

PROPERTY boPin172FaultRawValue : BOOL
GET
                    boPin172FaultRawValue := boPin172Fault.Value;

                  
END_GET
END_PROPERTY

PROPERTY boPin101FaultRawValue : BOOL
GET
                    boPin101FaultRawValue := boPin101Fault.Value;

                  
END_GET
END_PROPERTY

PROPERTY boPin125FaultRawValue : BOOL
GET
                    boPin125FaultRawValue := boPin125Fault.Value;

                  
END_GET
END_PROPERTY

PROPERTY boPin150FaultRawValue : BOOL
GET
                    boPin150FaultRawValue := boPin150Fault.Value;

                  
END_GET
END_PROPERTY

PROPERTY boPin174FaultRawValue : BOOL
GET
                    boPin174FaultRawValue := boPin174Fault.Value;

                  
END_GET
END_PROPERTY

PROPERTY boPin102FaultRawValue : BOOL
GET
                    boPin102FaultRawValue := boPin102Fault.Value;

                  
END_GET
END_PROPERTY

PROPERTY boPin126FaultRawValue : BOOL
GET
                    boPin126FaultRawValue := boPin126Fault.Value;

                  
END_GET
END_PROPERTY

PROPERTY boPin151FaultRawValue : BOOL
GET
                    boPin151FaultRawValue := boPin151Fault.Value;

                  
END_GET
END_PROPERTY

PROPERTY boPin175FaultRawValue : BOOL
GET
                    boPin175FaultRawValue := boPin175Fault.Value;

                  
END_GET
END_PROPERTY

PROPERTY boPin149FaultRawValue : BOOL
GET
                    boPin149FaultRawValue := boPin149Fault.Value;

                  
END_GET
END_PROPERTY

PROPERTY boPin173FaultRawValue : BOOL
GET
                    boPin173FaultRawValue := boPin173Fault.Value;

                  
END_GET
END_PROPERTY

PROPERTY boPin152FaultRawValue : BOOL
GET
                    boPin152FaultRawValue := boPin152Fault.Value;

                  
END_GET
END_PROPERTY

PROPERTY boPin176FaultRawValue : BOOL
GET
                    boPin176FaultRawValue := boPin176Fault.Value;

                  
END_GET
END_PROPERTY

PROPERTY boPin155FaultRawValue : BOOL
GET
                    boPin155FaultRawValue := boPin155Fault.Value;

                  
END_GET
END_PROPERTY

PROPERTY boPin179FaultRawValue : BOOL
GET
                    boPin179FaultRawValue := boPin179Fault.Value;

                  
END_GET
END_PROPERTY

PROPERTY boPin158FaultRawValue : BOOL
GET
                    boPin158FaultRawValue := boPin158Fault.Value;

                  
END_GET
END_PROPERTY

PROPERTY boPin182FaultRawValue : BOOL
GET
                    boPin182FaultRawValue := boPin182Fault.Value;

                  
END_GET
END_PROPERTY

PROPERTY boPin251FaultRawValue : BOOL
GET
                    boPin251FaultRawValue := boPin251Fault.Value;

                  
END_GET
END_PROPERTY

PROPERTY boPin238FaultRawValue : BOOL
GET
                    boPin238FaultRawValue := boPin238Fault.Value;

                  
END_GET
END_PROPERTY

PROPERTY boPin252FaultRawValue : BOOL
GET
                    boPin252FaultRawValue := boPin252Fault.Value;

                  
END_GET
END_PROPERTY

PROPERTY boPin239FaultRawValue : BOOL
GET
                    boPin239FaultRawValue := boPin239Fault.Value;

                  
END_GET
END_PROPERTY

PROPERTY boPin253FaultRawValue : BOOL
GET
                    boPin253FaultRawValue := boPin253Fault.Value;

                  
END_GET
END_PROPERTY

PROPERTY boPin240FaultRawValue : BOOL
GET
                    boPin240FaultRawValue := boPin240Fault.Value;

                  
END_GET
END_PROPERTY

PROPERTY boPin254FaultRawValue : BOOL
GET
                    boPin254FaultRawValue := boPin254Fault.Value;

                  
END_GET
END_PROPERTY

PROPERTY boPin241FaultRawValue : BOOL
GET
                    boPin241FaultRawValue := boPin241Fault.Value;

                  
END_GET
END_PROPERTY

PROPERTY boPin161FaultRawValue : BOOL
GET
                    boPin161FaultRawValue := boPin161Fault.Value;

                  
END_GET
END_PROPERTY

PROPERTY boPin185FaultRawValue : BOOL
GET
                    boPin185FaultRawValue := boPin185Fault.Value;

                  
END_GET
END_PROPERTY

PROPERTY boPin188FaultRawValue : BOOL
GET
                    boPin188FaultRawValue := boPin188Fault.Value;

                  
END_GET
END_PROPERTY

PROPERTY boPin164FaultRawValue : BOOL
GET
                    boPin164FaultRawValue := boPin164Fault.Value;

                  
END_GET
END_PROPERTY

PROPERTY boPin191FaultRawValue : BOOL
GET
                    boPin191FaultRawValue := boPin191Fault.Value;

                  
END_GET
END_PROPERTY

PROPERTY boPin167FaultRawValue : BOOL
GET
                    boPin167FaultRawValue := boPin167Fault.Value;

                  
END_GET
END_PROPERTY

PROPERTY boPin194FaultRawValue : BOOL
GET
                    boPin194FaultRawValue := boPin194Fault.Value;

                  
END_GET
END_PROPERTY

PROPERTY boPin170FaultRawValue : BOOL
GET
                    boPin170FaultRawValue := boPin170Fault.Value;

                  
END_GET
END_PROPERTY

PROPERTY boPin181FaultToolValue : BOOL
GET
                    boPin181FaultToolValue := boPin181Fault.Value;

                  
END_GET
END_PROPERTY

PROPERTY boPin160FaultToolValue : BOOL
GET
                    boPin160FaultToolValue := boPin160Fault.Value;

                  
END_GET
END_PROPERTY

PROPERTY boPin184FaultToolValue : BOOL
GET
                    boPin184FaultToolValue := boPin184Fault.Value;

                  
END_GET
END_PROPERTY

PROPERTY boPin187FaultToolValue : BOOL
GET
                    boPin187FaultToolValue := boPin187Fault.Value;

                  
END_GET
END_PROPERTY

PROPERTY boPin163FaultToolValue : BOOL
GET
                    boPin163FaultToolValue := boPin163Fault.Value;

                  
END_GET
END_PROPERTY

PROPERTY boPin190FaultToolValue : BOOL
GET
                    boPin190FaultToolValue := boPin190Fault.Value;

                  
END_GET
END_PROPERTY

PROPERTY boPin166FaultToolValue : BOOL
GET
                    boPin166FaultToolValue := boPin166Fault.Value;

                  
END_GET
END_PROPERTY

PROPERTY boPin193FaultToolValue : BOOL
GET
                    boPin193FaultToolValue := boPin193Fault.Value;

                  
END_GET
END_PROPERTY

PROPERTY boPin169FaultToolValue : BOOL
GET
                    boPin169FaultToolValue := boPin169Fault.Value;

                  
END_GET
END_PROPERTY

PROPERTY boPin196FaultToolValue : BOOL
GET
                    boPin196FaultToolValue := boPin196Fault.Value;

                  
END_GET
END_PROPERTY

PROPERTY boPin172FaultToolValue : BOOL
GET
                    boPin172FaultToolValue := boPin172Fault.Value;

                  
END_GET
END_PROPERTY

PROPERTY boPin101FaultToolValue : BOOL
GET
                    boPin101FaultToolValue := boPin101Fault.Value;

                  
END_GET
END_PROPERTY

PROPERTY boPin125FaultToolValue : BOOL
GET
                    boPin125FaultToolValue := boPin125Fault.Value;

                  
END_GET
END_PROPERTY

PROPERTY boPin150FaultToolValue : BOOL
GET
                    boPin150FaultToolValue := boPin150Fault.Value;

                  
END_GET
END_PROPERTY

PROPERTY boPin174FaultToolValue : BOOL
GET
                    boPin174FaultToolValue := boPin174Fault.Value;

                  
END_GET
END_PROPERTY

PROPERTY boPin102FaultToolValue : BOOL
GET
                    boPin102FaultToolValue := boPin102Fault.Value;

                  
END_GET
END_PROPERTY

PROPERTY boPin126FaultToolValue : BOOL
GET
                    boPin126FaultToolValue := boPin126Fault.Value;

                  
END_GET
END_PROPERTY

PROPERTY boPin151FaultToolValue : BOOL
GET
                    boPin151FaultToolValue := boPin151Fault.Value;

                  
END_GET
END_PROPERTY

PROPERTY boPin175FaultToolValue : BOOL
GET
                    boPin175FaultToolValue := boPin175Fault.Value;

                  
END_GET
END_PROPERTY

PROPERTY boPin149FaultToolValue : BOOL
GET
                    boPin149FaultToolValue := boPin149Fault.Value;

                  
END_GET
END_PROPERTY

PROPERTY boPin173FaultToolValue : BOOL
GET
                    boPin173FaultToolValue := boPin173Fault.Value;

                  
END_GET
END_PROPERTY

PROPERTY boPin152FaultToolValue : BOOL
GET
                    boPin152FaultToolValue := boPin152Fault.Value;

                  
END_GET
END_PROPERTY

PROPERTY boPin176FaultToolValue : BOOL
GET
                    boPin176FaultToolValue := boPin176Fault.Value;

                  
END_GET
END_PROPERTY

PROPERTY boPin155FaultToolValue : BOOL
GET
                    boPin155FaultToolValue := boPin155Fault.Value;

                  
END_GET
END_PROPERTY

PROPERTY boPin179FaultToolValue : BOOL
GET
                    boPin179FaultToolValue := boPin179Fault.Value;

                  
END_GET
END_PROPERTY

PROPERTY boPin158FaultToolValue : BOOL
GET
                    boPin158FaultToolValue := boPin158Fault.Value;

                  
END_GET
END_PROPERTY

PROPERTY boPin182FaultToolValue : BOOL
GET
                    boPin182FaultToolValue := boPin182Fault.Value;

                  
END_GET
END_PROPERTY

PROPERTY boPin251FaultToolValue : BOOL
GET
                    boPin251FaultToolValue := boPin251Fault.Value;

                  
END_GET
END_PROPERTY

PROPERTY boPin238FaultToolValue : BOOL
GET
                    boPin238FaultToolValue := boPin238Fault.Value;

                  
END_GET
END_PROPERTY

PROPERTY boPin252FaultToolValue : BOOL
GET
                    boPin252FaultToolValue := boPin252Fault.Value;

                  
END_GET
END_PROPERTY

PROPERTY boPin239FaultToolValue : BOOL
GET
                    boPin239FaultToolValue := boPin239Fault.Value;

                  
END_GET
END_PROPERTY

PROPERTY boPin253FaultToolValue : BOOL
GET
                    boPin253FaultToolValue := boPin253Fault.Value;

                  
END_GET
END_PROPERTY

PROPERTY boPin240FaultToolValue : BOOL
GET
                    boPin240FaultToolValue := boPin240Fault.Value;

                  
END_GET
END_PROPERTY

PROPERTY boPin254FaultToolValue : BOOL
GET
                    boPin254FaultToolValue := boPin254Fault.Value;

                  
END_GET
END_PROPERTY

PROPERTY boPin241FaultToolValue : BOOL
GET
                    boPin241FaultToolValue := boPin241Fault.Value;

                  
END_GET
END_PROPERTY

PROPERTY boPin161FaultToolValue : BOOL
GET
                    boPin161FaultToolValue := boPin161Fault.Value;

                  
END_GET
END_PROPERTY

PROPERTY boPin185FaultToolValue : BOOL
GET
                    boPin185FaultToolValue := boPin185Fault.Value;

                  
END_GET
END_PROPERTY

PROPERTY boPin188FaultToolValue : BOOL
GET
                    boPin188FaultToolValue := boPin188Fault.Value;

                  
END_GET
END_PROPERTY

PROPERTY boPin164FaultToolValue : BOOL
GET
                    boPin164FaultToolValue := boPin164Fault.Value;

                  
END_GET
END_PROPERTY

PROPERTY boPin191FaultToolValue : BOOL
GET
                    boPin191FaultToolValue := boPin191Fault.Value;

                  
END_GET
END_PROPERTY

PROPERTY boPin167FaultToolValue : BOOL
GET
                    boPin167FaultToolValue := boPin167Fault.Value;

                  
END_GET
END_PROPERTY

PROPERTY boPin194FaultToolValue : BOOL
GET
                    boPin194FaultToolValue := boPin194Fault.Value;

                  
END_GET
END_PROPERTY

PROPERTY boPin170FaultToolValue : BOOL
GET
                    boPin170FaultToolValue := boPin170Fault.Value;

                  
END_GET
END_PROPERTY

METHOD InitializeCanSignals
                  boPin181Fault.AppScalingDivisor :=1;
boPin181Fault.AppScalingMultiplier :=1;
boPin181Fault.AppScalingOffset :=0;
boPin181Fault.AppUnit :="";
boPin181Fault.CanDefault :=0;
boPin181Fault.CanInit :=0;
boPin181Fault.CanMax :=1;
boPin181Fault.CanMin :=0;
boPin181Fault.CanUnit :="";
boPin181Fault.Description :="for the Neotec diag pages";
boPin181Fault.ErrorReaction := eErrorReaction.ERSIG_DFLT;
boPin181Fault.ReceiverAdress :=1;
boPin181Fault.ToolScalingDivisor :=1;
boPin181Fault.ToolScalingMultiplier :=1;
boPin181Fault.ToolScalingOffset :=0;
boPin181Fault.ToolUnit :="";

boPin160Fault.AppScalingDivisor :=1;
boPin160Fault.AppScalingMultiplier :=1;
boPin160Fault.AppScalingOffset :=0;
boPin160Fault.AppUnit :="";
boPin160Fault.CanDefault :=0;
boPin160Fault.CanInit :=0;
boPin160Fault.CanMax :=1;
boPin160Fault.CanMin :=0;
boPin160Fault.CanUnit :="";
boPin160Fault.Description :="for the Neotec diag pages";
boPin160Fault.ErrorReaction := eErrorReaction.ERSIG_DFLT;
boPin160Fault.ReceiverAdress :=1;
boPin160Fault.ToolScalingDivisor :=1;
boPin160Fault.ToolScalingMultiplier :=1;
boPin160Fault.ToolScalingOffset :=0;
boPin160Fault.ToolUnit :="";

boPin184Fault.AppScalingDivisor :=1;
boPin184Fault.AppScalingMultiplier :=1;
boPin184Fault.AppScalingOffset :=0;
boPin184Fault.AppUnit :="";
boPin184Fault.CanDefault :=0;
boPin184Fault.CanInit :=0;
boPin184Fault.CanMax :=1;
boPin184Fault.CanMin :=0;
boPin184Fault.CanUnit :="";
boPin184Fault.Description :="for the Neotec diag pages";
boPin184Fault.ErrorReaction := eErrorReaction.ERSIG_DFLT;
boPin184Fault.ReceiverAdress :=1;
boPin184Fault.ToolScalingDivisor :=1;
boPin184Fault.ToolScalingMultiplier :=1;
boPin184Fault.ToolScalingOffset :=0;
boPin184Fault.ToolUnit :="";

boPin187Fault.AppScalingDivisor :=1;
boPin187Fault.AppScalingMultiplier :=1;
boPin187Fault.AppScalingOffset :=0;
boPin187Fault.AppUnit :="";
boPin187Fault.CanDefault :=0;
boPin187Fault.CanInit :=0;
boPin187Fault.CanMax :=1;
boPin187Fault.CanMin :=0;
boPin187Fault.CanUnit :="";
boPin187Fault.Description :="for the Neotec diag pages";
boPin187Fault.ErrorReaction := eErrorReaction.ERSIG_DFLT;
boPin187Fault.ReceiverAdress :=1;
boPin187Fault.ToolScalingDivisor :=1;
boPin187Fault.ToolScalingMultiplier :=1;
boPin187Fault.ToolScalingOffset :=0;
boPin187Fault.ToolUnit :="";

boPin163Fault.AppScalingDivisor :=1;
boPin163Fault.AppScalingMultiplier :=1;
boPin163Fault.AppScalingOffset :=0;
boPin163Fault.AppUnit :="";
boPin163Fault.CanDefault :=0;
boPin163Fault.CanInit :=0;
boPin163Fault.CanMax :=1;
boPin163Fault.CanMin :=0;
boPin163Fault.CanUnit :="";
boPin163Fault.Description :="for the Neotec diag pages";
boPin163Fault.ErrorReaction := eErrorReaction.ERSIG_DFLT;
boPin163Fault.ReceiverAdress :=1;
boPin163Fault.ToolScalingDivisor :=1;
boPin163Fault.ToolScalingMultiplier :=1;
boPin163Fault.ToolScalingOffset :=0;
boPin163Fault.ToolUnit :="";

boPin190Fault.AppScalingDivisor :=1;
boPin190Fault.AppScalingMultiplier :=1;
boPin190Fault.AppScalingOffset :=0;
boPin190Fault.AppUnit :="";
boPin190Fault.CanDefault :=0;
boPin190Fault.CanInit :=0;
boPin190Fault.CanMax :=1;
boPin190Fault.CanMin :=0;
boPin190Fault.CanUnit :="";
boPin190Fault.Description :="for the Neotec diag pages";
boPin190Fault.ErrorReaction := eErrorReaction.ERSIG_DFLT;
boPin190Fault.ReceiverAdress :=1;
boPin190Fault.ToolScalingDivisor :=1;
boPin190Fault.ToolScalingMultiplier :=1;
boPin190Fault.ToolScalingOffset :=0;
boPin190Fault.ToolUnit :="";

boPin166Fault.AppScalingDivisor :=1;
boPin166Fault.AppScalingMultiplier :=1;
boPin166Fault.AppScalingOffset :=0;
boPin166Fault.AppUnit :="";
boPin166Fault.CanDefault :=0;
boPin166Fault.CanInit :=0;
boPin166Fault.CanMax :=1;
boPin166Fault.CanMin :=0;
boPin166Fault.CanUnit :="";
boPin166Fault.Description :="for the Neotec diag pages";
boPin166Fault.ErrorReaction := eErrorReaction.ERSIG_DFLT;
boPin166Fault.ReceiverAdress :=1;
boPin166Fault.ToolScalingDivisor :=1;
boPin166Fault.ToolScalingMultiplier :=1;
boPin166Fault.ToolScalingOffset :=0;
boPin166Fault.ToolUnit :="";

